// TIA Portal V17 export
// export: Created 2025-03-05T08:02:58.0476046Z, ExportSetting WithDefaults, DisplayName Totally Integrated Automation Portal, DisplayVersion V17 Update 8, DisplayName TIA Portal Openness, DisplayVersion V17 Update 8, DisplayName TIA Portal Version Control Interface, DisplayVersion V17, DisplayName SINAMICS Startdrive Advanced, DisplayVersion V17 SP2, DisplayName SINAMICS Startdrive G110M, G120, G120C, G120D, G120P, G115D, DisplayVersion V17 SP2, DisplayName SINAMICS Startdrive G130, G150, S120, S150, SINAMICS MV, S210, DisplayVersion V17 SP2, DisplayName STEP 7 Professional, DisplayVersion V17 Update 8, DisplayName SINUMERIK ONE STEP 7 Toolbox, DisplayVersion V17 Update 12, DisplayName SINUMERIK 840D sl STEP 7 Toolbox, DisplayVersion V17 Update 12, DisplayName STEP 7 Safety, DisplayVersion V17 Update 6, DisplayName WinCC Advanced, DisplayVersion V17 Update 8
FUNCTION "FC16702_OPC_UA_MASTER_POWDER_DATA_UPDATE" : Void   // FC16702, LAD
{ S7_Optimized_Access := 'TRUE' }
VERSION : 0.1
// stored: AutoNumber false, IsIECCheckEnabled false, SetENOAutomatically false, UDAEnableTagReadback false
   VAR_TEMP
      CURRENT_1 : Real;
      CURRENT_2 : Real;
      CURRENT_3 : Real;
      CURRENT_4 : Real;
      CURRENT_5 : Real;
      CURRENT_6 : Real;
      CURRENT_7 : Real;
      CURRENT_8 : Real;
      CURRENT_9 : Real;
      CURRENT_10 : Real;
   END_VAR
BEGIN

REGION Network 1: <<<<<<<<<<<<<<<<<<<< OPC UA MASTER POWDER >>>>>>>>>>>>>>>>>>>>
END_REGION

REGION Network 2: <<<<<<<<<<<<<< GENERAL >>>>>>>>>>>>>>>>>>>>
END_REGION

REGION Network 3: GENERAL INFO
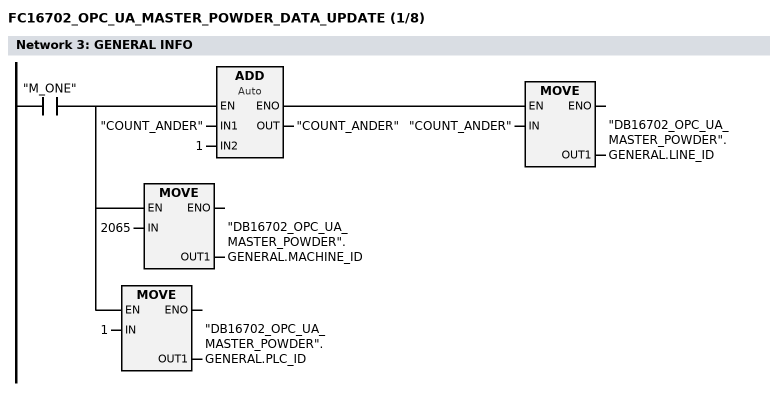
   RUNG wire#powerrail
      Contact( "M_ONE" )
      wire#w1
      Add(in1 := "COUNT_ANDER", in2 := 1, out => "COUNT_ANDER")
      Move(in := "COUNT_ANDER", out1 => "DB16702_OPC_UA_MASTER_POWDER".GENERAL.LINE_ID)
   END_RUNG
   RUNG wire#w1
      Move(in := 2065, out1 => "DB16702_OPC_UA_MASTER_POWDER".GENERAL.MACHINE_ID)
   END_RUNG
   RUNG wire#w1
      Move(in := 1, out1 => "DB16702_OPC_UA_MASTER_POWDER".GENERAL.PLC_ID)
   END_RUNG
   // the same network as SCL:
   IF "M_ONE" THEN
       "COUNT_ANDER" := "COUNT_ANDER" + 1;
       "DB16702_OPC_UA_MASTER_POWDER".GENERAL.LINE_ID := "COUNT_ANDER";
       "DB16702_OPC_UA_MASTER_POWDER".GENERAL.MACHINE_ID := 2065;
       "DB16702_OPC_UA_MASTER_POWDER".GENERAL.PLC_ID := 1;
   END_IF;
END_REGION

REGION Network 4: <<<<<<<<<<<<<< UNIT 01 >>>>>>>>>>>>>>>>>>>>
END_REGION

REGION Network 5: HOPPER 1 UNIT 01
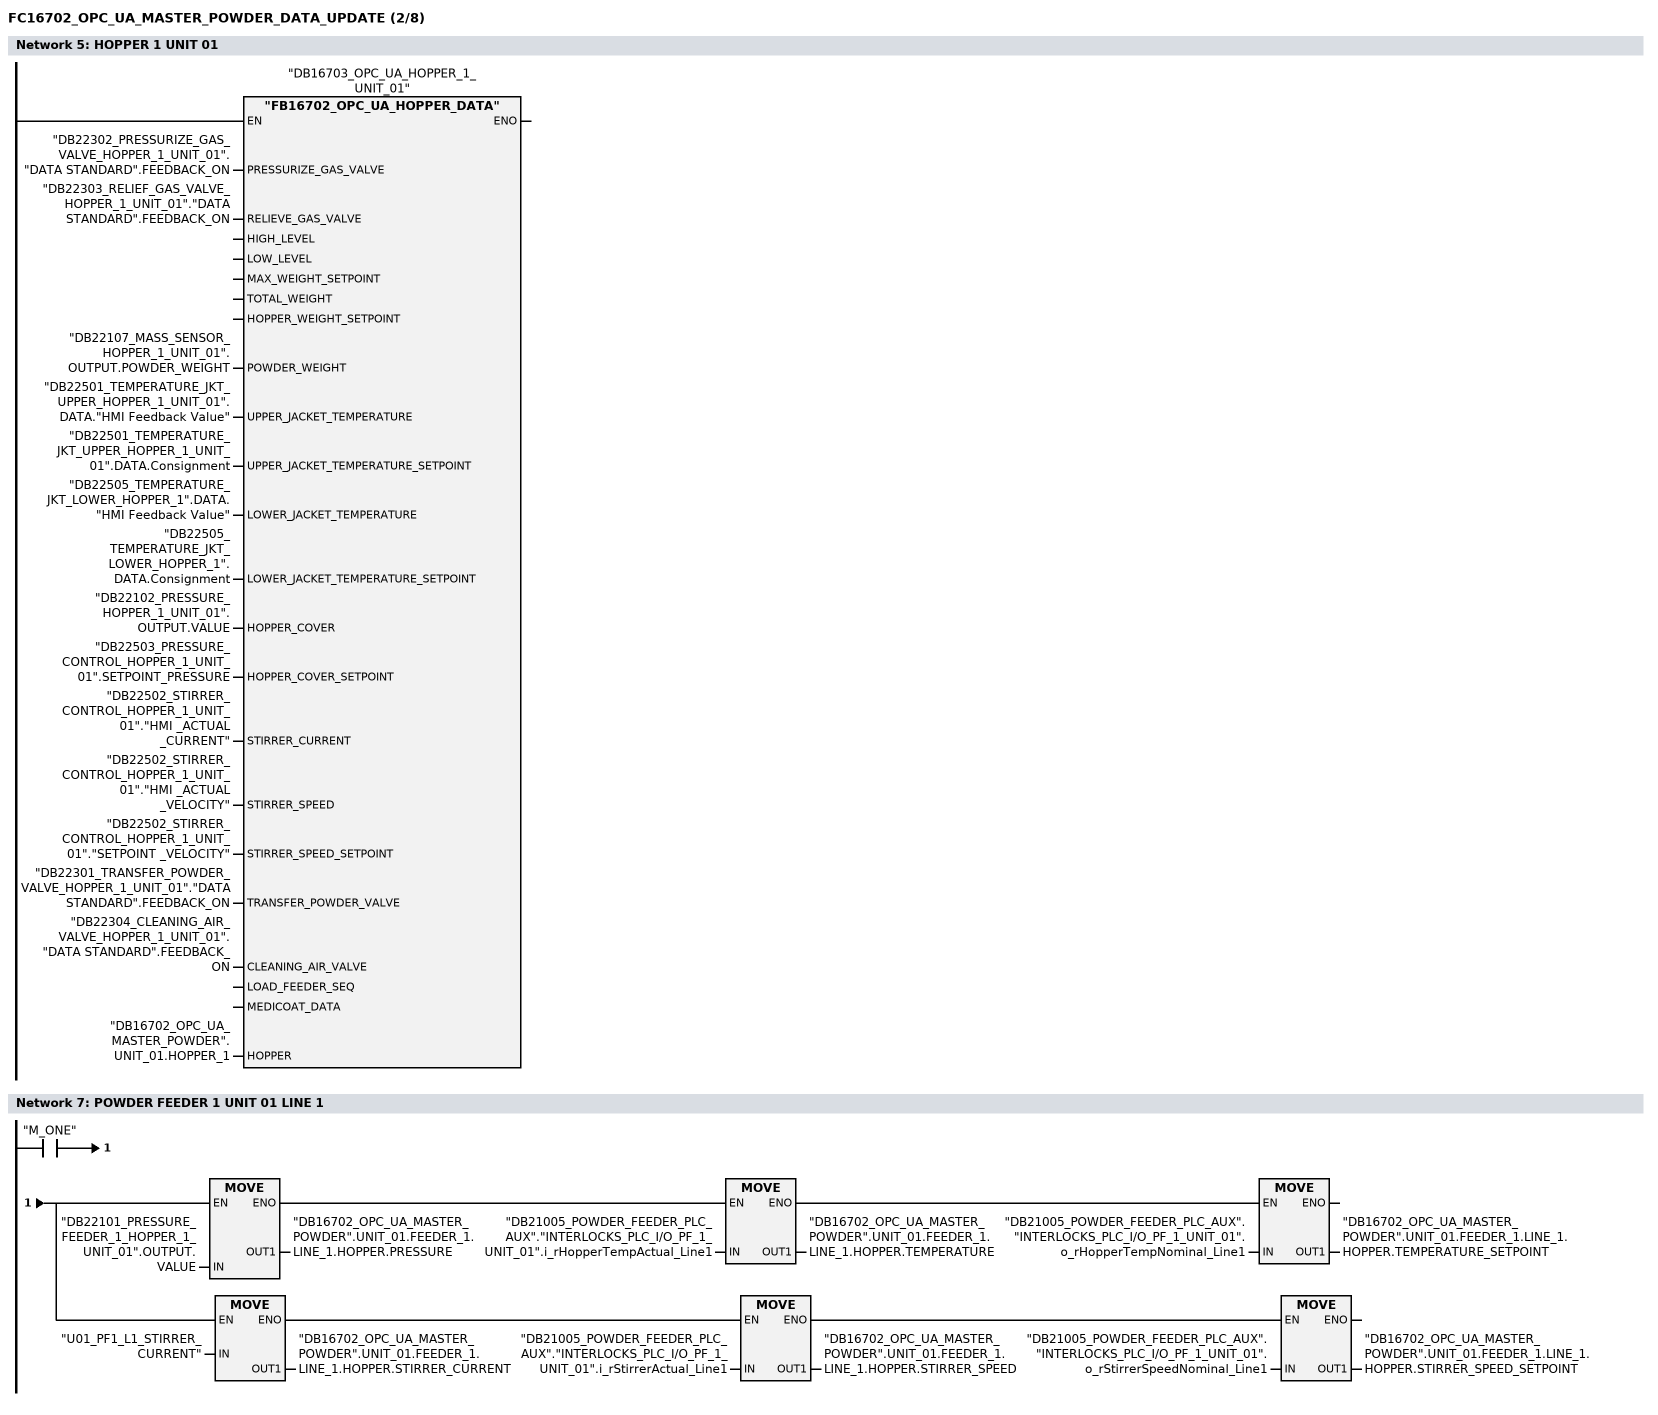
   RUNG wire#powerrail
      "DB16703_OPC_UA_HOPPER_1_UNIT_01"(PRESSURIZE_GAS_VALVE := "DB22302_PRESSURIZE_GAS_VALVE_HOPPER_1_UNIT_01"."DATA STANDARD".FEEDBACK_ON, RELIEVE_GAS_VALVE := "DB22303_RELIEF_GAS_VALVE_HOPPER_1_UNIT_01"."DATA STANDARD".FEEDBACK_ON, HIGH_LEVEL :=, LOW_LEVEL :=, MAX_WEIGHT_SETPOINT :=, TOTAL_WEIGHT :=, HOPPER_WEIGHT_SETPOINT :=, POWDER_WEIGHT := "DB22107_MASS_SENSOR_HOPPER_1_UNIT_01".OUTPUT.POWDER_WEIGHT, UPPER_JACKET_TEMPERATURE := "DB22501_TEMPERATURE_JKT_UPPER_HOPPER_1_UNIT_01".DATA."HMI Feedback Value", UPPER_JACKET_TEMPERATURE_SETPOINT := "DB22501_TEMPERATURE_JKT_UPPER_HOPPER_1_UNIT_01".DATA.Consignment, LOWER_JACKET_TEMPERATURE := "DB22505_TEMPERATURE_JKT_LOWER_HOPPER_1".DATA."HMI Feedback Value", LOWER_JACKET_TEMPERATURE_SETPOINT := "DB22505_TEMPERATURE_JKT_LOWER_HOPPER_1".DATA.Consignment, HOPPER_COVER := "DB22102_PRESSURE_HOPPER_1_UNIT_01".OUTPUT.VALUE, HOPPER_COVER_SETPOINT := "DB22503_PRESSURE_CONTROL_HOPPER_1_UNIT_01".SETPOINT_PRESSURE, STIRRER_CURRENT := "DB22502_STIRRER_CONTROL_HOPPER_1_UNIT_01"."HMI _ACTUAL _CURRENT", STIRRER_SPEED := "DB22502_STIRRER_CONTROL_HOPPER_1_UNIT_01"."HMI _ACTUAL _VELOCITY", STIRRER_SPEED_SETPOINT := "DB22502_STIRRER_CONTROL_HOPPER_1_UNIT_01"."SETPOINT _VELOCITY", TRANSFER_POWDER_VALVE := "DB22301_TRANSFER_POWDER_VALVE_HOPPER_1_UNIT_01"."DATA STANDARD".FEEDBACK_ON, CLEANING_AIR_VALVE := "DB22304_CLEANING_AIR_VALVE_HOPPER_1_UNIT_01"."DATA STANDARD".FEEDBACK_ON, LOAD_FEEDER_SEQ :=, MEDICOAT_DATA :=, HOPPER := "DB16702_OPC_UA_MASTER_POWDER".UNIT_01.HOPPER_1)
   END_RUNG
   // the same network as SCL:
   "DB16703_OPC_UA_HOPPER_1_UNIT_01"(PRESSURIZE_GAS_VALVE := "DB22302_PRESSURIZE_GAS_VALVE_HOPPER_1_UNIT_01"."DATA STANDARD".FEEDBACK_ON,   // "FB16702_OPC_UA_HOPPER_DATA"
                           RELIEVE_GAS_VALVE := "DB22303_RELIEF_GAS_VALVE_HOPPER_1_UNIT_01"."DATA STANDARD".FEEDBACK_ON,
                           POWDER_WEIGHT := "DB22107_MASS_SENSOR_HOPPER_1_UNIT_01".OUTPUT.POWDER_WEIGHT,
                           UPPER_JACKET_TEMPERATURE := "DB22501_TEMPERATURE_JKT_UPPER_HOPPER_1_UNIT_01".DATA."HMI Feedback Value",
                           UPPER_JACKET_TEMPERATURE_SETPOINT := "DB22501_TEMPERATURE_JKT_UPPER_HOPPER_1_UNIT_01".DATA.Consignment,
                           LOWER_JACKET_TEMPERATURE := "DB22505_TEMPERATURE_JKT_LOWER_HOPPER_1".DATA."HMI Feedback Value",
                           LOWER_JACKET_TEMPERATURE_SETPOINT := "DB22505_TEMPERATURE_JKT_LOWER_HOPPER_1".DATA.Consignment,
                           HOPPER_COVER := "DB22102_PRESSURE_HOPPER_1_UNIT_01".OUTPUT.VALUE,
                           HOPPER_COVER_SETPOINT := "DB22503_PRESSURE_CONTROL_HOPPER_1_UNIT_01".SETPOINT_PRESSURE,
                           STIRRER_CURRENT := "DB22502_STIRRER_CONTROL_HOPPER_1_UNIT_01"."HMI _ACTUAL _CURRENT",
                           STIRRER_SPEED := "DB22502_STIRRER_CONTROL_HOPPER_1_UNIT_01"."HMI _ACTUAL _VELOCITY",
                           STIRRER_SPEED_SETPOINT := "DB22502_STIRRER_CONTROL_HOPPER_1_UNIT_01"."SETPOINT _VELOCITY",
                           TRANSFER_POWDER_VALVE := "DB22301_TRANSFER_POWDER_VALVE_HOPPER_1_UNIT_01"."DATA STANDARD".FEEDBACK_ON,
                           CLEANING_AIR_VALVE := "DB22304_CLEANING_AIR_VALVE_HOPPER_1_UNIT_01"."DATA STANDARD".FEEDBACK_ON,
                           HOPPER := "DB16702_OPC_UA_MASTER_POWDER".UNIT_01.HOPPER_1);
END_REGION

REGION Network 6: HOPPER 2 UNIT 01
END_REGION

REGION Network 7: POWDER FEEDER 1 UNIT 01 LINE 1
   RUNG wire#powerrail
      Contact( "M_ONE" )
      wire#w1
      Move(in := "DB22101_PRESSURE_FEEDER_1_HOPPER_1_UNIT_01".OUTPUT.VALUE, out1 => "DB16702_OPC_UA_MASTER_POWDER".UNIT_01.FEEDER_1.LINE_1.HOPPER.PRESSURE)
      Move(in := "DB21005_POWDER_FEEDER_PLC_AUX"."INTERLOCKS_PLC_I/O_PF_1_UNIT_01".i_rHopperTempActual_Line1, out1 => "DB16702_OPC_UA_MASTER_POWDER".UNIT_01.FEEDER_1.LINE_1.HOPPER.TEMPERATURE)
      Move(in := "DB21005_POWDER_FEEDER_PLC_AUX"."INTERLOCKS_PLC_I/O_PF_1_UNIT_01".o_rHopperTempNominal_Line1, out1 => "DB16702_OPC_UA_MASTER_POWDER".UNIT_01.FEEDER_1.LINE_1.HOPPER.TEMPERATURE_SETPOINT)
   END_RUNG
   RUNG wire#w1
      Move(in := "U01_PF1_L1_STIRRER_CURRENT", out1 => "DB16702_OPC_UA_MASTER_POWDER".UNIT_01.FEEDER_1.LINE_1.HOPPER.STIRRER_CURRENT)
      Move(in := "DB21005_POWDER_FEEDER_PLC_AUX"."INTERLOCKS_PLC_I/O_PF_1_UNIT_01".i_rStirrerActual_Line1, out1 => "DB16702_OPC_UA_MASTER_POWDER".UNIT_01.FEEDER_1.LINE_1.HOPPER.STIRRER_SPEED)
      Move(in := "DB21005_POWDER_FEEDER_PLC_AUX"."INTERLOCKS_PLC_I/O_PF_1_UNIT_01".o_rStirrerSpeedNominal_Line1, out1 => "DB16702_OPC_UA_MASTER_POWDER".UNIT_01.FEEDER_1.LINE_1.HOPPER.STIRRER_SPEED_SETPOINT)
   END_RUNG
   // the same network as SCL:
   IF "M_ONE" THEN
       "DB16702_OPC_UA_MASTER_POWDER".UNIT_01.FEEDER_1.LINE_1.HOPPER.PRESSURE := "DB22101_PRESSURE_FEEDER_1_HOPPER_1_UNIT_01".OUTPUT.VALUE;
       "DB16702_OPC_UA_MASTER_POWDER".UNIT_01.FEEDER_1.LINE_1.HOPPER.TEMPERATURE := "DB21005_POWDER_FEEDER_PLC_AUX"."INTERLOCKS_PLC_I/O_PF_1_UNIT_01".i_rHopperTempActual_Line1;
       "DB16702_OPC_UA_MASTER_POWDER".UNIT_01.FEEDER_1.LINE_1.HOPPER.TEMPERATURE_SETPOINT := "DB21005_POWDER_FEEDER_PLC_AUX"."INTERLOCKS_PLC_I/O_PF_1_UNIT_01".o_rHopperTempNominal_Line1;
       "DB16702_OPC_UA_MASTER_POWDER".UNIT_01.FEEDER_1.LINE_1.HOPPER.STIRRER_CURRENT := "U01_PF1_L1_STIRRER_CURRENT";
       "DB16702_OPC_UA_MASTER_POWDER".UNIT_01.FEEDER_1.LINE_1.HOPPER.STIRRER_SPEED := "DB21005_POWDER_FEEDER_PLC_AUX"."INTERLOCKS_PLC_I/O_PF_1_UNIT_01".i_rStirrerActual_Line1;
       "DB16702_OPC_UA_MASTER_POWDER".UNIT_01.FEEDER_1.LINE_1.HOPPER.STIRRER_SPEED_SETPOINT := "DB21005_POWDER_FEEDER_PLC_AUX"."INTERLOCKS_PLC_I/O_PF_1_UNIT_01".o_rStirrerSpeedNominal_Line1;
   END_IF;
END_REGION

REGION Network 8: POWDER FEEDER 1 UNIT 01 LINE 1 DISK
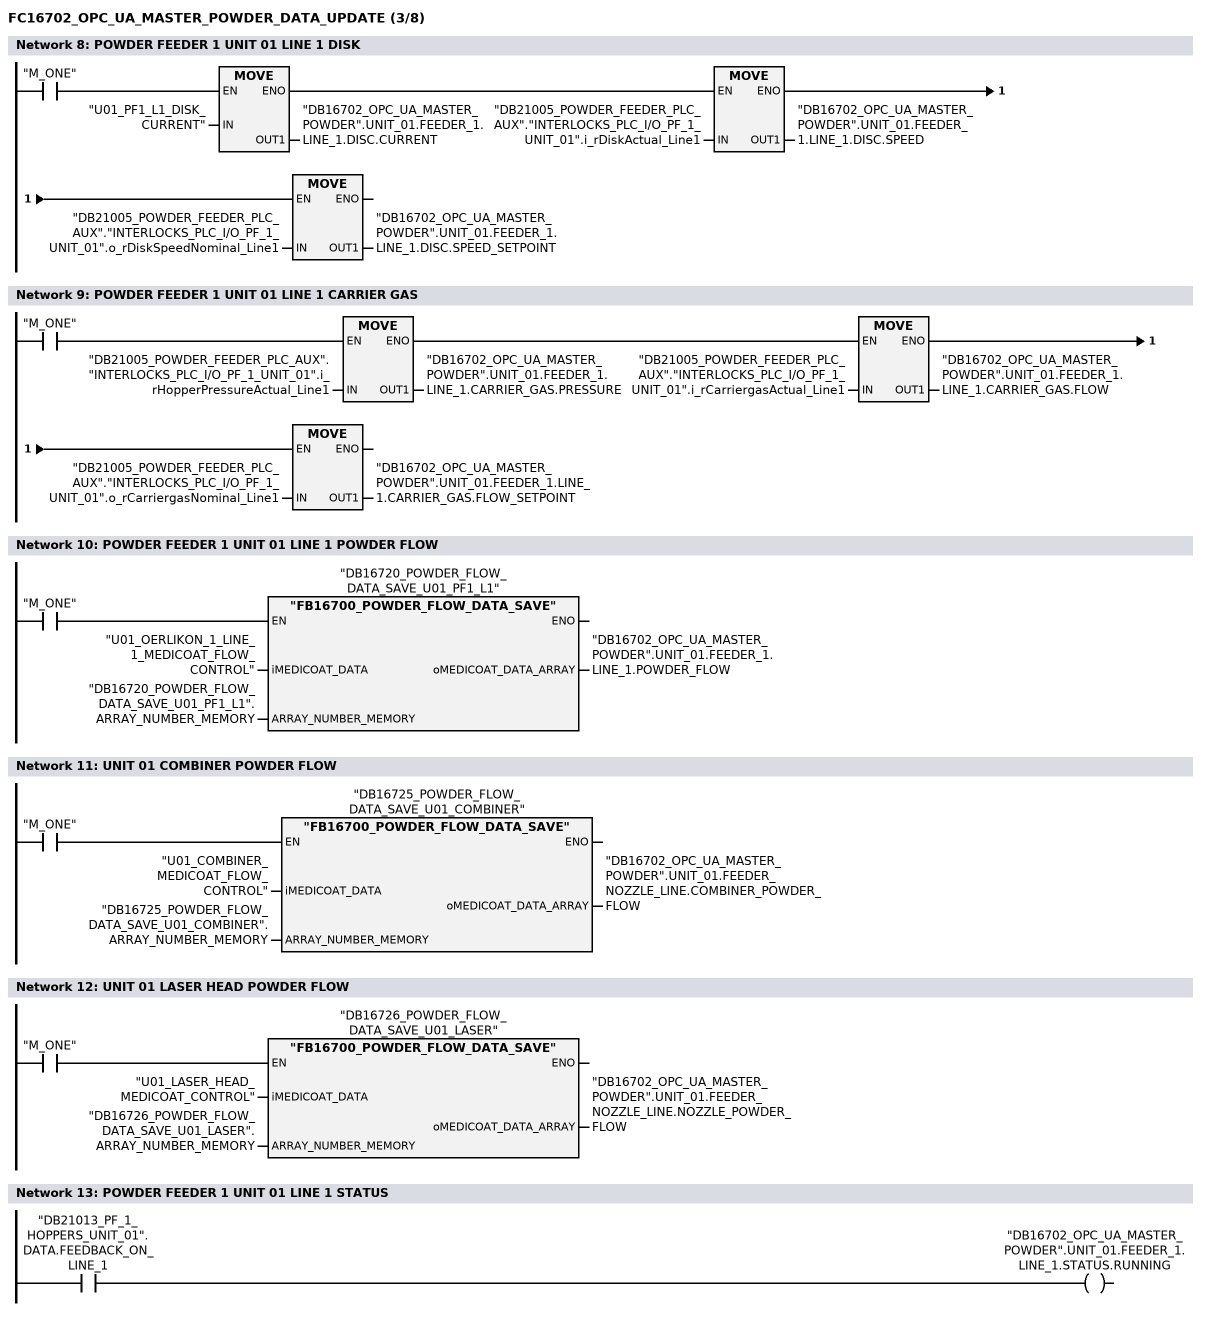
   RUNG wire#powerrail
      Contact( "M_ONE" )
      Move(in := "U01_PF1_L1_DISK_CURRENT", out1 => "DB16702_OPC_UA_MASTER_POWDER".UNIT_01.FEEDER_1.LINE_1.DISC.CURRENT)
      Move(in := "DB21005_POWDER_FEEDER_PLC_AUX"."INTERLOCKS_PLC_I/O_PF_1_UNIT_01".i_rDiskActual_Line1, out1 => "DB16702_OPC_UA_MASTER_POWDER".UNIT_01.FEEDER_1.LINE_1.DISC.SPEED)
      Move(in := "DB21005_POWDER_FEEDER_PLC_AUX"."INTERLOCKS_PLC_I/O_PF_1_UNIT_01".o_rDiskSpeedNominal_Line1, out1 => "DB16702_OPC_UA_MASTER_POWDER".UNIT_01.FEEDER_1.LINE_1.DISC.SPEED_SETPOINT)
   END_RUNG
   // the same network as SCL:
   IF "M_ONE" THEN
       "DB16702_OPC_UA_MASTER_POWDER".UNIT_01.FEEDER_1.LINE_1.DISC.CURRENT := "U01_PF1_L1_DISK_CURRENT";
       "DB16702_OPC_UA_MASTER_POWDER".UNIT_01.FEEDER_1.LINE_1.DISC.SPEED := "DB21005_POWDER_FEEDER_PLC_AUX"."INTERLOCKS_PLC_I/O_PF_1_UNIT_01".i_rDiskActual_Line1;
       "DB16702_OPC_UA_MASTER_POWDER".UNIT_01.FEEDER_1.LINE_1.DISC.SPEED_SETPOINT := "DB21005_POWDER_FEEDER_PLC_AUX"."INTERLOCKS_PLC_I/O_PF_1_UNIT_01".o_rDiskSpeedNominal_Line1;
   END_IF;
END_REGION

REGION Network 9: POWDER FEEDER 1 UNIT 01 LINE 1 CARRIER GAS
   RUNG wire#powerrail
      Contact( "M_ONE" )
      Move(in := "DB21005_POWDER_FEEDER_PLC_AUX"."INTERLOCKS_PLC_I/O_PF_1_UNIT_01".i_rHopperPressureActual_Line1, out1 => "DB16702_OPC_UA_MASTER_POWDER".UNIT_01.FEEDER_1.LINE_1.CARRIER_GAS.PRESSURE)
      Move(in := "DB21005_POWDER_FEEDER_PLC_AUX"."INTERLOCKS_PLC_I/O_PF_1_UNIT_01".i_rCarriergasActual_Line1, out1 => "DB16702_OPC_UA_MASTER_POWDER".UNIT_01.FEEDER_1.LINE_1.CARRIER_GAS.FLOW)
      Move(in := "DB21005_POWDER_FEEDER_PLC_AUX"."INTERLOCKS_PLC_I/O_PF_1_UNIT_01".o_rCarriergasNominal_Line1, out1 => "DB16702_OPC_UA_MASTER_POWDER".UNIT_01.FEEDER_1.LINE_1.CARRIER_GAS.FLOW_SETPOINT)
   END_RUNG
   // the same network as SCL:
   IF "M_ONE" THEN
       "DB16702_OPC_UA_MASTER_POWDER".UNIT_01.FEEDER_1.LINE_1.CARRIER_GAS.PRESSURE := "DB21005_POWDER_FEEDER_PLC_AUX"."INTERLOCKS_PLC_I/O_PF_1_UNIT_01".i_rHopperPressureActual_Line1;
       "DB16702_OPC_UA_MASTER_POWDER".UNIT_01.FEEDER_1.LINE_1.CARRIER_GAS.FLOW := "DB21005_POWDER_FEEDER_PLC_AUX"."INTERLOCKS_PLC_I/O_PF_1_UNIT_01".i_rCarriergasActual_Line1;
       "DB16702_OPC_UA_MASTER_POWDER".UNIT_01.FEEDER_1.LINE_1.CARRIER_GAS.FLOW_SETPOINT := "DB21005_POWDER_FEEDER_PLC_AUX"."INTERLOCKS_PLC_I/O_PF_1_UNIT_01".o_rCarriergasNominal_Line1;
   END_IF;
END_REGION

REGION Network 10: POWDER FEEDER 1 UNIT 01 LINE 1 POWDER FLOW
   RUNG wire#powerrail
      Contact( "M_ONE" )
      "DB16720_POWDER_FLOW_DATA_SAVE_U01_PF1_L1"(iMEDICOAT_DATA := "U01_OERLIKON_1_LINE_1_MEDICOAT_FLOW_CONTROL", ARRAY_NUMBER_MEMORY := "DB16720_POWDER_FLOW_DATA_SAVE_U01_PF1_L1".ARRAY_NUMBER_MEMORY, oMEDICOAT_DATA_ARRAY => "DB16702_OPC_UA_MASTER_POWDER".UNIT_01.FEEDER_1.LINE_1.POWDER_FLOW)
   END_RUNG
   // the same network as SCL:
   IF "M_ONE" THEN
       "DB16720_POWDER_FLOW_DATA_SAVE_U01_PF1_L1"(iMEDICOAT_DATA := "U01_OERLIKON_1_LINE_1_MEDICOAT_FLOW_CONTROL",   // "FB16700_POWDER_FLOW_DATA_SAVE"
                               ARRAY_NUMBER_MEMORY := "DB16720_POWDER_FLOW_DATA_SAVE_U01_PF1_L1".ARRAY_NUMBER_MEMORY,
                               oMEDICOAT_DATA_ARRAY => "DB16702_OPC_UA_MASTER_POWDER".UNIT_01.FEEDER_1.LINE_1.POWDER_FLOW);
   END_IF;
END_REGION

REGION Network 11: UNIT 01 COMBINER POWDER FLOW
   RUNG wire#powerrail
      Contact( "M_ONE" )
      "DB16725_POWDER_FLOW_DATA_SAVE_U01_COMBINER"(iMEDICOAT_DATA := "U01_COMBINER_MEDICOAT_FLOW_CONTROL", ARRAY_NUMBER_MEMORY := "DB16725_POWDER_FLOW_DATA_SAVE_U01_COMBINER".ARRAY_NUMBER_MEMORY, oMEDICOAT_DATA_ARRAY => "DB16702_OPC_UA_MASTER_POWDER".UNIT_01.FEEDER_NOZZLE_LINE.COMBINER_POWDER_FLOW)
   END_RUNG
   // the same network as SCL:
   IF "M_ONE" THEN
       "DB16725_POWDER_FLOW_DATA_SAVE_U01_COMBINER"(iMEDICOAT_DATA := "U01_COMBINER_MEDICOAT_FLOW_CONTROL",   // "FB16700_POWDER_FLOW_DATA_SAVE"
                               ARRAY_NUMBER_MEMORY := "DB16725_POWDER_FLOW_DATA_SAVE_U01_COMBINER".ARRAY_NUMBER_MEMORY,
                               oMEDICOAT_DATA_ARRAY => "DB16702_OPC_UA_MASTER_POWDER".UNIT_01.FEEDER_NOZZLE_LINE.COMBINER_POWDER_FLOW);
   END_IF;
END_REGION

REGION Network 12: UNIT 01 LASER HEAD POWDER FLOW
   RUNG wire#powerrail
      Contact( "M_ONE" )
      "DB16726_POWDER_FLOW_DATA_SAVE_U01_LASER"(iMEDICOAT_DATA := "U01_LASER_HEAD_MEDICOAT_CONTROL", ARRAY_NUMBER_MEMORY := "DB16726_POWDER_FLOW_DATA_SAVE_U01_LASER".ARRAY_NUMBER_MEMORY, oMEDICOAT_DATA_ARRAY => "DB16702_OPC_UA_MASTER_POWDER".UNIT_01.FEEDER_NOZZLE_LINE.NOZZLE_POWDER_FLOW)
   END_RUNG
   // the same network as SCL:
   IF "M_ONE" THEN
       "DB16726_POWDER_FLOW_DATA_SAVE_U01_LASER"(iMEDICOAT_DATA := "U01_LASER_HEAD_MEDICOAT_CONTROL",   // "FB16700_POWDER_FLOW_DATA_SAVE"
                               ARRAY_NUMBER_MEMORY := "DB16726_POWDER_FLOW_DATA_SAVE_U01_LASER".ARRAY_NUMBER_MEMORY,
                               oMEDICOAT_DATA_ARRAY => "DB16702_OPC_UA_MASTER_POWDER".UNIT_01.FEEDER_NOZZLE_LINE.NOZZLE_POWDER_FLOW);
   END_IF;
END_REGION

REGION Network 13: POWDER FEEDER 1 UNIT 01 LINE 1 STATUS
   RUNG wire#powerrail
      Contact( "DB21013_PF_1_HOPPERS_UNIT_01".DATA.FEEDBACK_ON_LINE_1 )
      Coil( "DB16702_OPC_UA_MASTER_POWDER".UNIT_01.FEEDER_1.LINE_1.STATUS.RUNNING )
   END_RUNG
   // the same network as SCL:
   "DB16702_OPC_UA_MASTER_POWDER".UNIT_01.FEEDER_1.LINE_1.STATUS.RUNNING := "DB21013_PF_1_HOPPERS_UNIT_01".DATA.FEEDBACK_ON_LINE_1;
END_REGION

REGION Network 14: POWDER FEEDER 1 UNIT 01 LINE 2 HOPPER
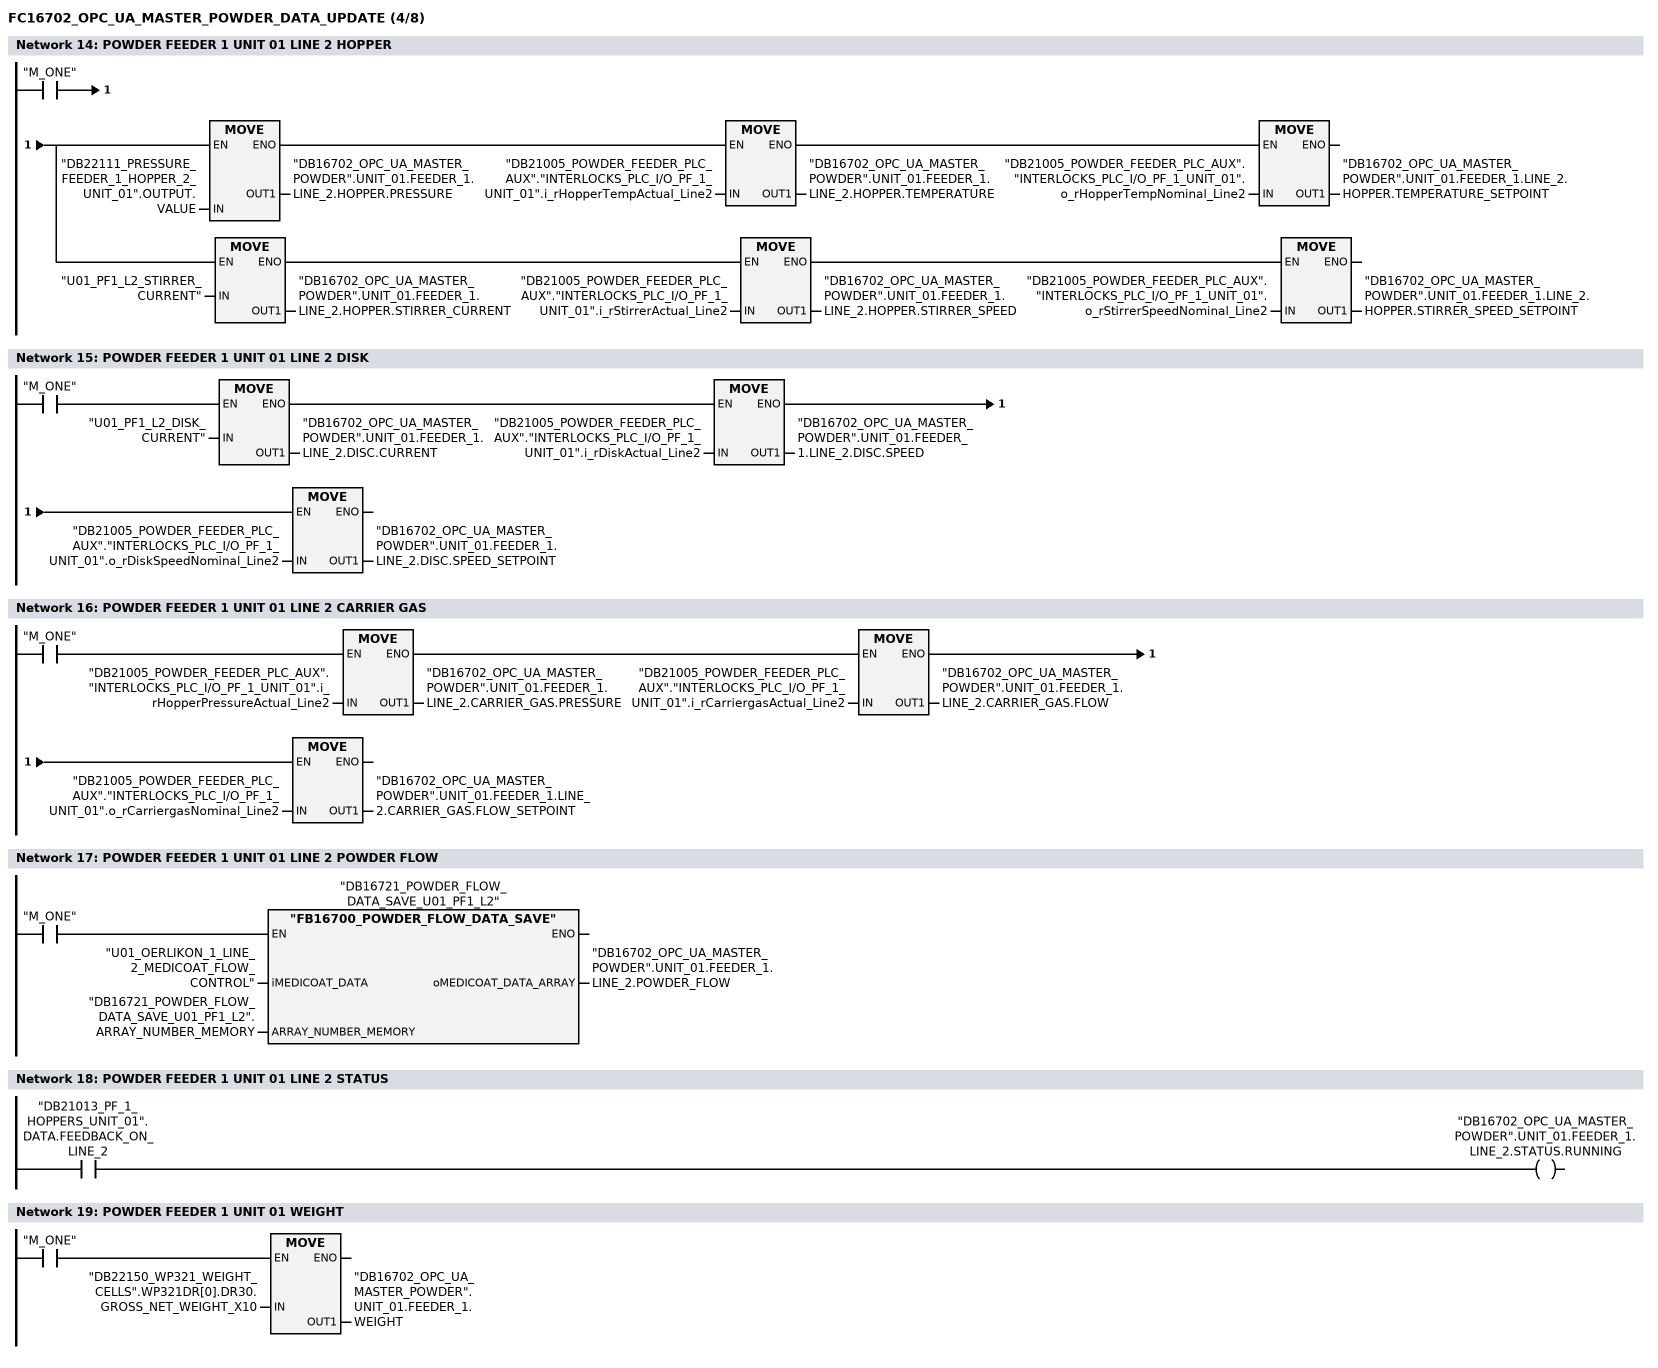
   RUNG wire#powerrail
      Contact( "M_ONE" )
      wire#w1
      Move(in := "DB22111_PRESSURE_FEEDER_1_HOPPER_2_UNIT_01".OUTPUT.VALUE, out1 => "DB16702_OPC_UA_MASTER_POWDER".UNIT_01.FEEDER_1.LINE_2.HOPPER.PRESSURE)
      Move(in := "DB21005_POWDER_FEEDER_PLC_AUX"."INTERLOCKS_PLC_I/O_PF_1_UNIT_01".i_rHopperTempActual_Line2, out1 => "DB16702_OPC_UA_MASTER_POWDER".UNIT_01.FEEDER_1.LINE_2.HOPPER.TEMPERATURE)
      Move(in := "DB21005_POWDER_FEEDER_PLC_AUX"."INTERLOCKS_PLC_I/O_PF_1_UNIT_01".o_rHopperTempNominal_Line2, out1 => "DB16702_OPC_UA_MASTER_POWDER".UNIT_01.FEEDER_1.LINE_2.HOPPER.TEMPERATURE_SETPOINT)
   END_RUNG
   RUNG wire#w1
      Move(in := "U01_PF1_L2_STIRRER_CURRENT", out1 => "DB16702_OPC_UA_MASTER_POWDER".UNIT_01.FEEDER_1.LINE_2.HOPPER.STIRRER_CURRENT)
      Move(in := "DB21005_POWDER_FEEDER_PLC_AUX"."INTERLOCKS_PLC_I/O_PF_1_UNIT_01".i_rStirrerActual_Line2, out1 => "DB16702_OPC_UA_MASTER_POWDER".UNIT_01.FEEDER_1.LINE_2.HOPPER.STIRRER_SPEED)
      Move(in := "DB21005_POWDER_FEEDER_PLC_AUX"."INTERLOCKS_PLC_I/O_PF_1_UNIT_01".o_rStirrerSpeedNominal_Line2, out1 => "DB16702_OPC_UA_MASTER_POWDER".UNIT_01.FEEDER_1.LINE_2.HOPPER.STIRRER_SPEED_SETPOINT)
   END_RUNG
   // the same network as SCL:
   IF "M_ONE" THEN
       "DB16702_OPC_UA_MASTER_POWDER".UNIT_01.FEEDER_1.LINE_2.HOPPER.PRESSURE := "DB22111_PRESSURE_FEEDER_1_HOPPER_2_UNIT_01".OUTPUT.VALUE;
       "DB16702_OPC_UA_MASTER_POWDER".UNIT_01.FEEDER_1.LINE_2.HOPPER.TEMPERATURE := "DB21005_POWDER_FEEDER_PLC_AUX"."INTERLOCKS_PLC_I/O_PF_1_UNIT_01".i_rHopperTempActual_Line2;
       "DB16702_OPC_UA_MASTER_POWDER".UNIT_01.FEEDER_1.LINE_2.HOPPER.TEMPERATURE_SETPOINT := "DB21005_POWDER_FEEDER_PLC_AUX"."INTERLOCKS_PLC_I/O_PF_1_UNIT_01".o_rHopperTempNominal_Line2;
       "DB16702_OPC_UA_MASTER_POWDER".UNIT_01.FEEDER_1.LINE_2.HOPPER.STIRRER_CURRENT := "U01_PF1_L2_STIRRER_CURRENT";
       "DB16702_OPC_UA_MASTER_POWDER".UNIT_01.FEEDER_1.LINE_2.HOPPER.STIRRER_SPEED := "DB21005_POWDER_FEEDER_PLC_AUX"."INTERLOCKS_PLC_I/O_PF_1_UNIT_01".i_rStirrerActual_Line2;
       "DB16702_OPC_UA_MASTER_POWDER".UNIT_01.FEEDER_1.LINE_2.HOPPER.STIRRER_SPEED_SETPOINT := "DB21005_POWDER_FEEDER_PLC_AUX"."INTERLOCKS_PLC_I/O_PF_1_UNIT_01".o_rStirrerSpeedNominal_Line2;
   END_IF;
END_REGION

REGION Network 15: POWDER FEEDER 1 UNIT 01 LINE 2 DISK
   RUNG wire#powerrail
      Contact( "M_ONE" )
      Move(in := "U01_PF1_L2_DISK_CURRENT", out1 => "DB16702_OPC_UA_MASTER_POWDER".UNIT_01.FEEDER_1.LINE_2.DISC.CURRENT)
      Move(in := "DB21005_POWDER_FEEDER_PLC_AUX"."INTERLOCKS_PLC_I/O_PF_1_UNIT_01".i_rDiskActual_Line2, out1 => "DB16702_OPC_UA_MASTER_POWDER".UNIT_01.FEEDER_1.LINE_2.DISC.SPEED)
      Move(in := "DB21005_POWDER_FEEDER_PLC_AUX"."INTERLOCKS_PLC_I/O_PF_1_UNIT_01".o_rDiskSpeedNominal_Line2, out1 => "DB16702_OPC_UA_MASTER_POWDER".UNIT_01.FEEDER_1.LINE_2.DISC.SPEED_SETPOINT)
   END_RUNG
   // the same network as SCL:
   IF "M_ONE" THEN
       "DB16702_OPC_UA_MASTER_POWDER".UNIT_01.FEEDER_1.LINE_2.DISC.CURRENT := "U01_PF1_L2_DISK_CURRENT";
       "DB16702_OPC_UA_MASTER_POWDER".UNIT_01.FEEDER_1.LINE_2.DISC.SPEED := "DB21005_POWDER_FEEDER_PLC_AUX"."INTERLOCKS_PLC_I/O_PF_1_UNIT_01".i_rDiskActual_Line2;
       "DB16702_OPC_UA_MASTER_POWDER".UNIT_01.FEEDER_1.LINE_2.DISC.SPEED_SETPOINT := "DB21005_POWDER_FEEDER_PLC_AUX"."INTERLOCKS_PLC_I/O_PF_1_UNIT_01".o_rDiskSpeedNominal_Line2;
   END_IF;
END_REGION

REGION Network 16: POWDER FEEDER 1 UNIT 01 LINE 2 CARRIER GAS
   RUNG wire#powerrail
      Contact( "M_ONE" )
      Move(in := "DB21005_POWDER_FEEDER_PLC_AUX"."INTERLOCKS_PLC_I/O_PF_1_UNIT_01".i_rHopperPressureActual_Line2, out1 => "DB16702_OPC_UA_MASTER_POWDER".UNIT_01.FEEDER_1.LINE_2.CARRIER_GAS.PRESSURE)
      Move(in := "DB21005_POWDER_FEEDER_PLC_AUX"."INTERLOCKS_PLC_I/O_PF_1_UNIT_01".i_rCarriergasActual_Line2, out1 => "DB16702_OPC_UA_MASTER_POWDER".UNIT_01.FEEDER_1.LINE_2.CARRIER_GAS.FLOW)
      Move(in := "DB21005_POWDER_FEEDER_PLC_AUX"."INTERLOCKS_PLC_I/O_PF_1_UNIT_01".o_rCarriergasNominal_Line2, out1 => "DB16702_OPC_UA_MASTER_POWDER".UNIT_01.FEEDER_1.LINE_2.CARRIER_GAS.FLOW_SETPOINT)
   END_RUNG
   // the same network as SCL:
   IF "M_ONE" THEN
       "DB16702_OPC_UA_MASTER_POWDER".UNIT_01.FEEDER_1.LINE_2.CARRIER_GAS.PRESSURE := "DB21005_POWDER_FEEDER_PLC_AUX"."INTERLOCKS_PLC_I/O_PF_1_UNIT_01".i_rHopperPressureActual_Line2;
       "DB16702_OPC_UA_MASTER_POWDER".UNIT_01.FEEDER_1.LINE_2.CARRIER_GAS.FLOW := "DB21005_POWDER_FEEDER_PLC_AUX"."INTERLOCKS_PLC_I/O_PF_1_UNIT_01".i_rCarriergasActual_Line2;
       "DB16702_OPC_UA_MASTER_POWDER".UNIT_01.FEEDER_1.LINE_2.CARRIER_GAS.FLOW_SETPOINT := "DB21005_POWDER_FEEDER_PLC_AUX"."INTERLOCKS_PLC_I/O_PF_1_UNIT_01".o_rCarriergasNominal_Line2;
   END_IF;
END_REGION

REGION Network 17: POWDER FEEDER 1 UNIT 01 LINE 2 POWDER FLOW
   RUNG wire#powerrail
      Contact( "M_ONE" )
      "DB16721_POWDER_FLOW_DATA_SAVE_U01_PF1_L2"(iMEDICOAT_DATA := "U01_OERLIKON_1_LINE_2_MEDICOAT_FLOW_CONTROL", ARRAY_NUMBER_MEMORY := "DB16721_POWDER_FLOW_DATA_SAVE_U01_PF1_L2".ARRAY_NUMBER_MEMORY, oMEDICOAT_DATA_ARRAY => "DB16702_OPC_UA_MASTER_POWDER".UNIT_01.FEEDER_1.LINE_2.POWDER_FLOW)
   END_RUNG
   // the same network as SCL:
   IF "M_ONE" THEN
       "DB16721_POWDER_FLOW_DATA_SAVE_U01_PF1_L2"(iMEDICOAT_DATA := "U01_OERLIKON_1_LINE_2_MEDICOAT_FLOW_CONTROL",   // "FB16700_POWDER_FLOW_DATA_SAVE"
                               ARRAY_NUMBER_MEMORY := "DB16721_POWDER_FLOW_DATA_SAVE_U01_PF1_L2".ARRAY_NUMBER_MEMORY,
                               oMEDICOAT_DATA_ARRAY => "DB16702_OPC_UA_MASTER_POWDER".UNIT_01.FEEDER_1.LINE_2.POWDER_FLOW);
   END_IF;
END_REGION

REGION Network 18: POWDER FEEDER 1 UNIT 01 LINE 2 STATUS
   RUNG wire#powerrail
      Contact( "DB21013_PF_1_HOPPERS_UNIT_01".DATA.FEEDBACK_ON_LINE_2 )
      Coil( "DB16702_OPC_UA_MASTER_POWDER".UNIT_01.FEEDER_1.LINE_2.STATUS.RUNNING )
   END_RUNG
   // the same network as SCL:
   "DB16702_OPC_UA_MASTER_POWDER".UNIT_01.FEEDER_1.LINE_2.STATUS.RUNNING := "DB21013_PF_1_HOPPERS_UNIT_01".DATA.FEEDBACK_ON_LINE_2;
END_REGION

REGION Network 19: POWDER FEEDER 1 UNIT 01 WEIGHT
   RUNG wire#powerrail
      Contact( "M_ONE" )
      Move(in := "DB22150_WP321_WEIGHT_CELLS".WP321DR[0].DR30.GROSS_NET_WEIGHT_X10, out1 => "DB16702_OPC_UA_MASTER_POWDER".UNIT_01.FEEDER_1.WEIGHT)
   END_RUNG
   // the same network as SCL:
   IF "M_ONE" THEN
       "DB16702_OPC_UA_MASTER_POWDER".UNIT_01.FEEDER_1.WEIGHT := "DB22150_WP321_WEIGHT_CELLS".WP321DR[0].DR30.GROSS_NET_WEIGHT_X10;
   END_IF;
END_REGION

REGION Network 20: <<<<<<<<<<<<<< UNIT 02 >>>>>>>>>>>>>>>>>>>>
END_REGION

REGION Network 21: POWDER FEEDER 1 UNIT 02 LINE 1 HOPPER
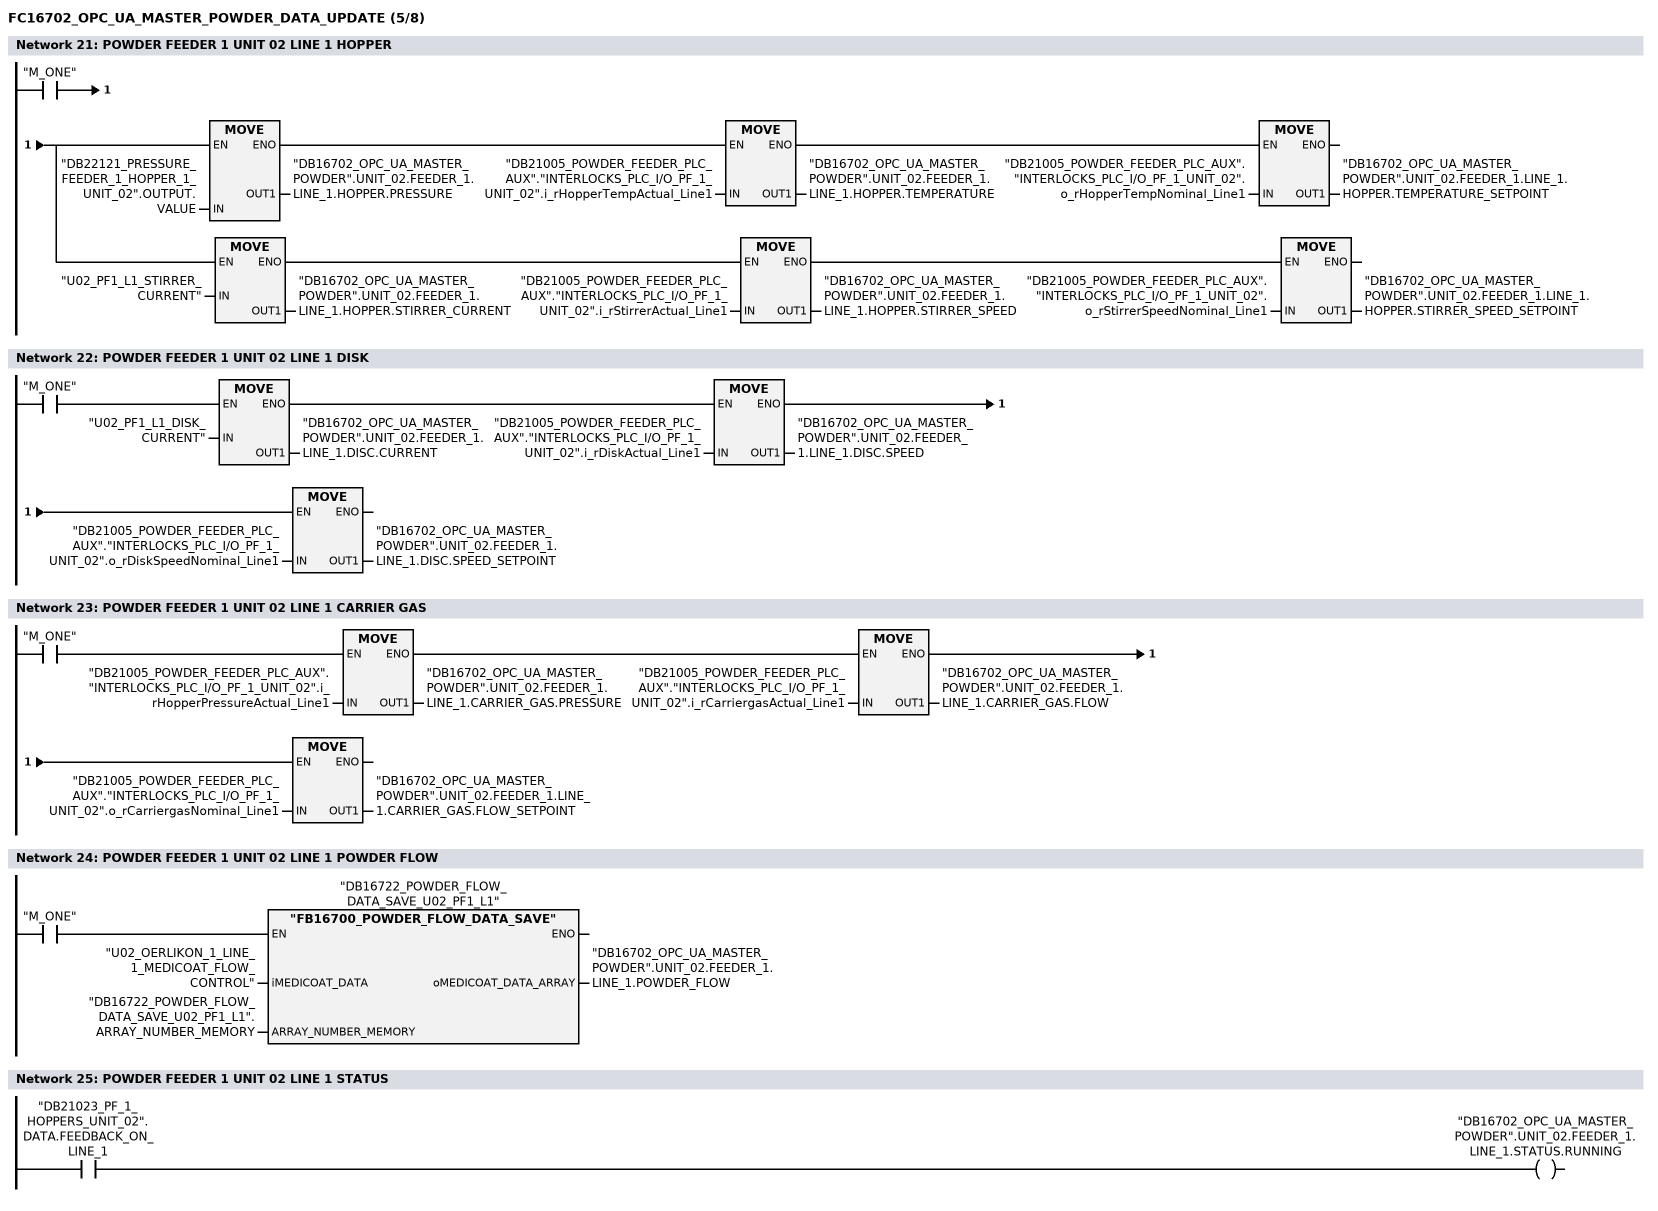
   RUNG wire#powerrail
      Contact( "M_ONE" )
      wire#w1
      Move(in := "DB22121_PRESSURE_FEEDER_1_HOPPER_1_UNIT_02".OUTPUT.VALUE, out1 => "DB16702_OPC_UA_MASTER_POWDER".UNIT_02.FEEDER_1.LINE_1.HOPPER.PRESSURE)
      Move(in := "DB21005_POWDER_FEEDER_PLC_AUX"."INTERLOCKS_PLC_I/O_PF_1_UNIT_02".i_rHopperTempActual_Line1, out1 => "DB16702_OPC_UA_MASTER_POWDER".UNIT_02.FEEDER_1.LINE_1.HOPPER.TEMPERATURE)
      Move(in := "DB21005_POWDER_FEEDER_PLC_AUX"."INTERLOCKS_PLC_I/O_PF_1_UNIT_02".o_rHopperTempNominal_Line1, out1 => "DB16702_OPC_UA_MASTER_POWDER".UNIT_02.FEEDER_1.LINE_1.HOPPER.TEMPERATURE_SETPOINT)
   END_RUNG
   RUNG wire#w1
      Move(in := "U02_PF1_L1_STIRRER_CURRENT", out1 => "DB16702_OPC_UA_MASTER_POWDER".UNIT_02.FEEDER_1.LINE_1.HOPPER.STIRRER_CURRENT)
      Move(in := "DB21005_POWDER_FEEDER_PLC_AUX"."INTERLOCKS_PLC_I/O_PF_1_UNIT_02".i_rStirrerActual_Line1, out1 => "DB16702_OPC_UA_MASTER_POWDER".UNIT_02.FEEDER_1.LINE_1.HOPPER.STIRRER_SPEED)
      Move(in := "DB21005_POWDER_FEEDER_PLC_AUX"."INTERLOCKS_PLC_I/O_PF_1_UNIT_02".o_rStirrerSpeedNominal_Line1, out1 => "DB16702_OPC_UA_MASTER_POWDER".UNIT_02.FEEDER_1.LINE_1.HOPPER.STIRRER_SPEED_SETPOINT)
   END_RUNG
   // the same network as SCL:
   IF "M_ONE" THEN
       "DB16702_OPC_UA_MASTER_POWDER".UNIT_02.FEEDER_1.LINE_1.HOPPER.PRESSURE := "DB22121_PRESSURE_FEEDER_1_HOPPER_1_UNIT_02".OUTPUT.VALUE;
       "DB16702_OPC_UA_MASTER_POWDER".UNIT_02.FEEDER_1.LINE_1.HOPPER.TEMPERATURE := "DB21005_POWDER_FEEDER_PLC_AUX"."INTERLOCKS_PLC_I/O_PF_1_UNIT_02".i_rHopperTempActual_Line1;
       "DB16702_OPC_UA_MASTER_POWDER".UNIT_02.FEEDER_1.LINE_1.HOPPER.TEMPERATURE_SETPOINT := "DB21005_POWDER_FEEDER_PLC_AUX"."INTERLOCKS_PLC_I/O_PF_1_UNIT_02".o_rHopperTempNominal_Line1;
       "DB16702_OPC_UA_MASTER_POWDER".UNIT_02.FEEDER_1.LINE_1.HOPPER.STIRRER_CURRENT := "U02_PF1_L1_STIRRER_CURRENT";
       "DB16702_OPC_UA_MASTER_POWDER".UNIT_02.FEEDER_1.LINE_1.HOPPER.STIRRER_SPEED := "DB21005_POWDER_FEEDER_PLC_AUX"."INTERLOCKS_PLC_I/O_PF_1_UNIT_02".i_rStirrerActual_Line1;
       "DB16702_OPC_UA_MASTER_POWDER".UNIT_02.FEEDER_1.LINE_1.HOPPER.STIRRER_SPEED_SETPOINT := "DB21005_POWDER_FEEDER_PLC_AUX"."INTERLOCKS_PLC_I/O_PF_1_UNIT_02".o_rStirrerSpeedNominal_Line1;
   END_IF;
END_REGION

REGION Network 22: POWDER FEEDER 1 UNIT 02 LINE 1 DISK
   RUNG wire#powerrail
      Contact( "M_ONE" )
      Move(in := "U02_PF1_L1_DISK_CURRENT", out1 => "DB16702_OPC_UA_MASTER_POWDER".UNIT_02.FEEDER_1.LINE_1.DISC.CURRENT)
      Move(in := "DB21005_POWDER_FEEDER_PLC_AUX"."INTERLOCKS_PLC_I/O_PF_1_UNIT_02".i_rDiskActual_Line1, out1 => "DB16702_OPC_UA_MASTER_POWDER".UNIT_02.FEEDER_1.LINE_1.DISC.SPEED)
      Move(in := "DB21005_POWDER_FEEDER_PLC_AUX"."INTERLOCKS_PLC_I/O_PF_1_UNIT_02".o_rDiskSpeedNominal_Line1, out1 => "DB16702_OPC_UA_MASTER_POWDER".UNIT_02.FEEDER_1.LINE_1.DISC.SPEED_SETPOINT)
   END_RUNG
   // the same network as SCL:
   IF "M_ONE" THEN
       "DB16702_OPC_UA_MASTER_POWDER".UNIT_02.FEEDER_1.LINE_1.DISC.CURRENT := "U02_PF1_L1_DISK_CURRENT";
       "DB16702_OPC_UA_MASTER_POWDER".UNIT_02.FEEDER_1.LINE_1.DISC.SPEED := "DB21005_POWDER_FEEDER_PLC_AUX"."INTERLOCKS_PLC_I/O_PF_1_UNIT_02".i_rDiskActual_Line1;
       "DB16702_OPC_UA_MASTER_POWDER".UNIT_02.FEEDER_1.LINE_1.DISC.SPEED_SETPOINT := "DB21005_POWDER_FEEDER_PLC_AUX"."INTERLOCKS_PLC_I/O_PF_1_UNIT_02".o_rDiskSpeedNominal_Line1;
   END_IF;
END_REGION

REGION Network 23: POWDER FEEDER 1 UNIT 02 LINE 1 CARRIER GAS
   RUNG wire#powerrail
      Contact( "M_ONE" )
      Move(in := "DB21005_POWDER_FEEDER_PLC_AUX"."INTERLOCKS_PLC_I/O_PF_1_UNIT_02".i_rHopperPressureActual_Line1, out1 => "DB16702_OPC_UA_MASTER_POWDER".UNIT_02.FEEDER_1.LINE_1.CARRIER_GAS.PRESSURE)
      Move(in := "DB21005_POWDER_FEEDER_PLC_AUX"."INTERLOCKS_PLC_I/O_PF_1_UNIT_02".i_rCarriergasActual_Line1, out1 => "DB16702_OPC_UA_MASTER_POWDER".UNIT_02.FEEDER_1.LINE_1.CARRIER_GAS.FLOW)
      Move(in := "DB21005_POWDER_FEEDER_PLC_AUX"."INTERLOCKS_PLC_I/O_PF_1_UNIT_02".o_rCarriergasNominal_Line1, out1 => "DB16702_OPC_UA_MASTER_POWDER".UNIT_02.FEEDER_1.LINE_1.CARRIER_GAS.FLOW_SETPOINT)
   END_RUNG
   // the same network as SCL:
   IF "M_ONE" THEN
       "DB16702_OPC_UA_MASTER_POWDER".UNIT_02.FEEDER_1.LINE_1.CARRIER_GAS.PRESSURE := "DB21005_POWDER_FEEDER_PLC_AUX"."INTERLOCKS_PLC_I/O_PF_1_UNIT_02".i_rHopperPressureActual_Line1;
       "DB16702_OPC_UA_MASTER_POWDER".UNIT_02.FEEDER_1.LINE_1.CARRIER_GAS.FLOW := "DB21005_POWDER_FEEDER_PLC_AUX"."INTERLOCKS_PLC_I/O_PF_1_UNIT_02".i_rCarriergasActual_Line1;
       "DB16702_OPC_UA_MASTER_POWDER".UNIT_02.FEEDER_1.LINE_1.CARRIER_GAS.FLOW_SETPOINT := "DB21005_POWDER_FEEDER_PLC_AUX"."INTERLOCKS_PLC_I/O_PF_1_UNIT_02".o_rCarriergasNominal_Line1;
   END_IF;
END_REGION

REGION Network 24: POWDER FEEDER 1 UNIT 02 LINE 1 POWDER FLOW
   RUNG wire#powerrail
      Contact( "M_ONE" )
      "DB16722_POWDER_FLOW_DATA_SAVE_U02_PF1_L1"(iMEDICOAT_DATA := "U02_OERLIKON_1_LINE_1_MEDICOAT_FLOW_CONTROL", ARRAY_NUMBER_MEMORY := "DB16722_POWDER_FLOW_DATA_SAVE_U02_PF1_L1".ARRAY_NUMBER_MEMORY, oMEDICOAT_DATA_ARRAY => "DB16702_OPC_UA_MASTER_POWDER".UNIT_02.FEEDER_1.LINE_1.POWDER_FLOW)
   END_RUNG
   // the same network as SCL:
   IF "M_ONE" THEN
       "DB16722_POWDER_FLOW_DATA_SAVE_U02_PF1_L1"(iMEDICOAT_DATA := "U02_OERLIKON_1_LINE_1_MEDICOAT_FLOW_CONTROL",   // "FB16700_POWDER_FLOW_DATA_SAVE"
                               ARRAY_NUMBER_MEMORY := "DB16722_POWDER_FLOW_DATA_SAVE_U02_PF1_L1".ARRAY_NUMBER_MEMORY,
                               oMEDICOAT_DATA_ARRAY => "DB16702_OPC_UA_MASTER_POWDER".UNIT_02.FEEDER_1.LINE_1.POWDER_FLOW);
   END_IF;
END_REGION

REGION Network 25: POWDER FEEDER 1 UNIT 02 LINE 1 STATUS
   RUNG wire#powerrail
      Contact( "DB21023_PF_1_HOPPERS_UNIT_02".DATA.FEEDBACK_ON_LINE_1 )
      Coil( "DB16702_OPC_UA_MASTER_POWDER".UNIT_02.FEEDER_1.LINE_1.STATUS.RUNNING )
   END_RUNG
   // the same network as SCL:
   "DB16702_OPC_UA_MASTER_POWDER".UNIT_02.FEEDER_1.LINE_1.STATUS.RUNNING := "DB21023_PF_1_HOPPERS_UNIT_02".DATA.FEEDBACK_ON_LINE_1;
END_REGION

REGION Network 26: POWDER FEEDER 1 UNIT 02 LINE 2 HOPPER
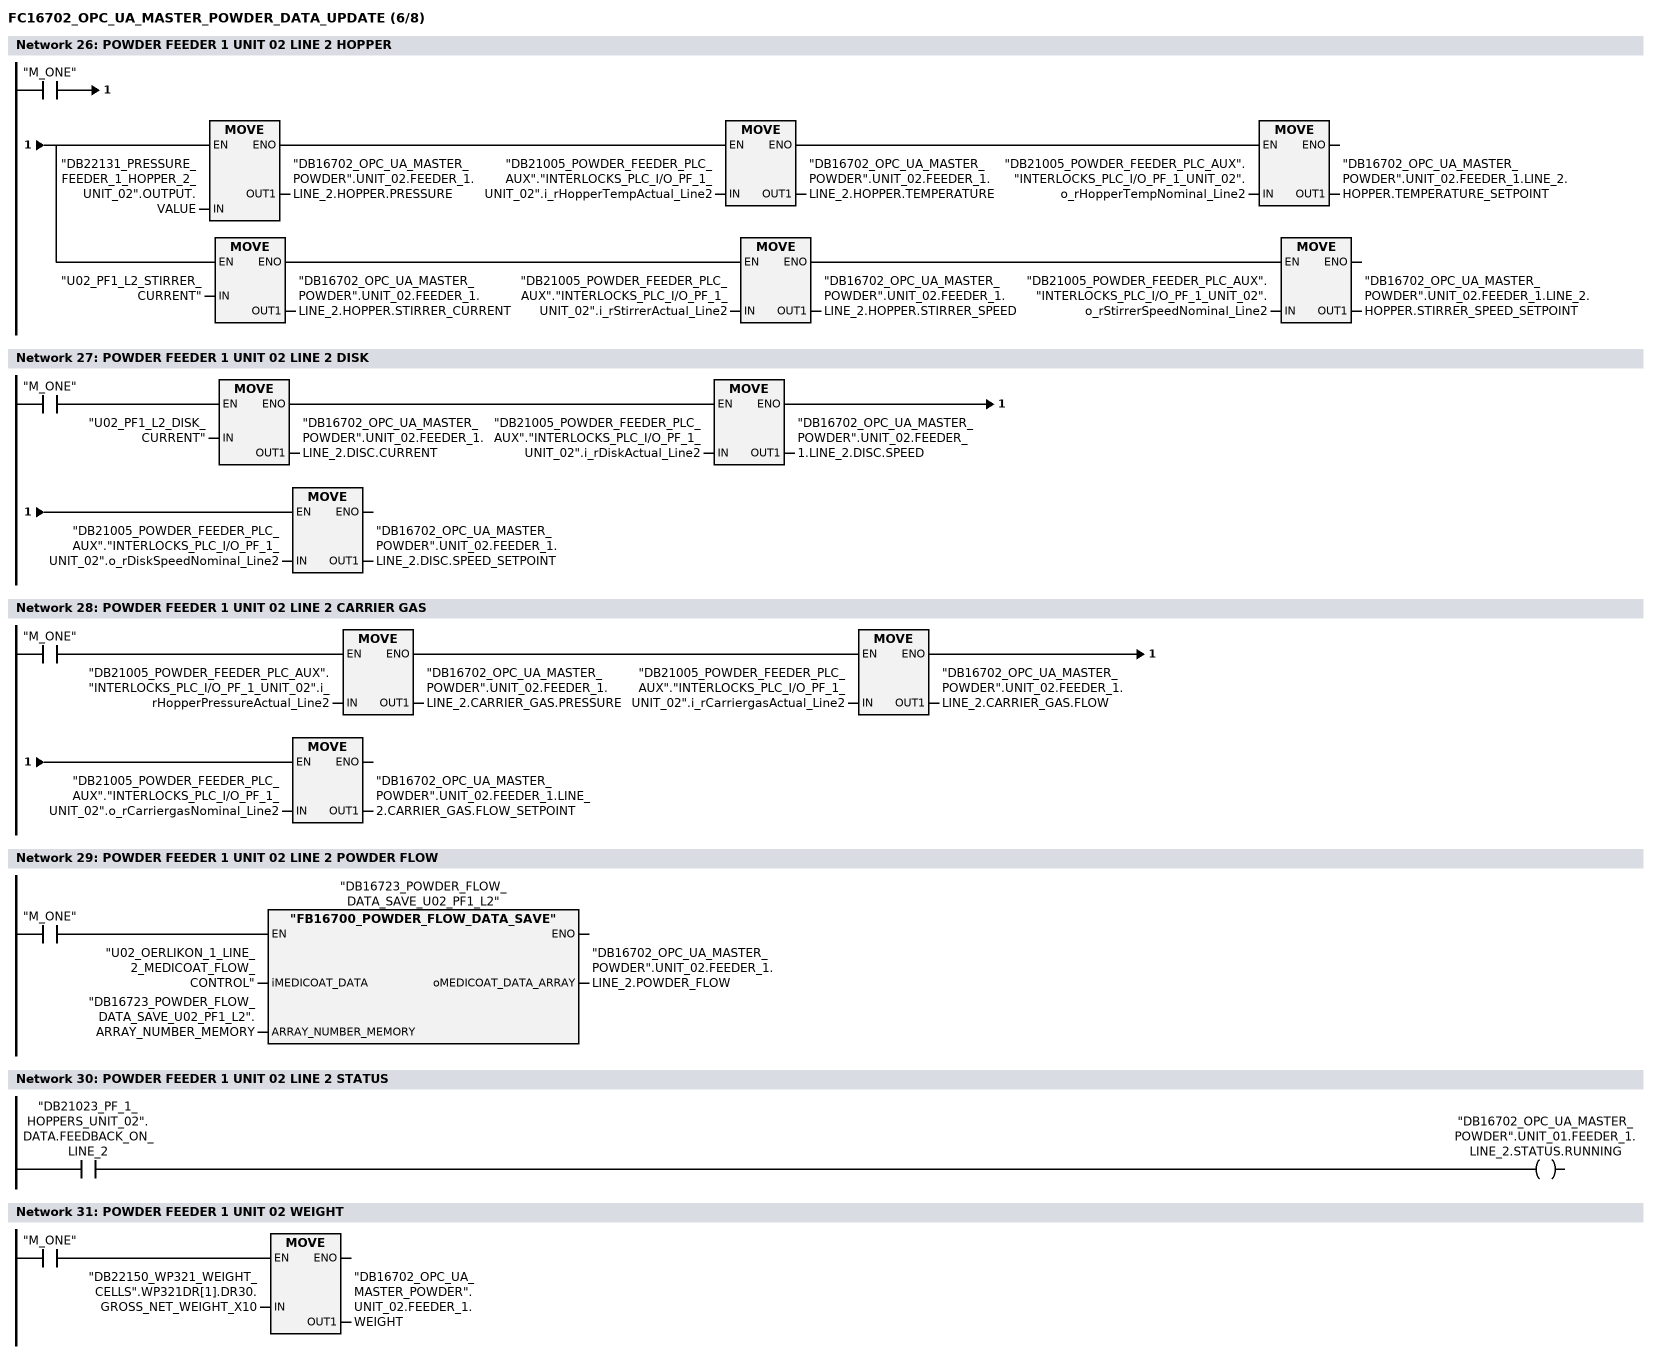
   RUNG wire#powerrail
      Contact( "M_ONE" )
      wire#w1
      Move(in := "DB22131_PRESSURE_FEEDER_1_HOPPER_2_UNIT_02".OUTPUT.VALUE, out1 => "DB16702_OPC_UA_MASTER_POWDER".UNIT_02.FEEDER_1.LINE_2.HOPPER.PRESSURE)
      Move(in := "DB21005_POWDER_FEEDER_PLC_AUX"."INTERLOCKS_PLC_I/O_PF_1_UNIT_02".i_rHopperTempActual_Line2, out1 => "DB16702_OPC_UA_MASTER_POWDER".UNIT_02.FEEDER_1.LINE_2.HOPPER.TEMPERATURE)
      Move(in := "DB21005_POWDER_FEEDER_PLC_AUX"."INTERLOCKS_PLC_I/O_PF_1_UNIT_02".o_rHopperTempNominal_Line2, out1 => "DB16702_OPC_UA_MASTER_POWDER".UNIT_02.FEEDER_1.LINE_2.HOPPER.TEMPERATURE_SETPOINT)
   END_RUNG
   RUNG wire#w1
      Move(in := "U02_PF1_L2_STIRRER_CURRENT", out1 => "DB16702_OPC_UA_MASTER_POWDER".UNIT_02.FEEDER_1.LINE_2.HOPPER.STIRRER_CURRENT)
      Move(in := "DB21005_POWDER_FEEDER_PLC_AUX"."INTERLOCKS_PLC_I/O_PF_1_UNIT_02".i_rStirrerActual_Line2, out1 => "DB16702_OPC_UA_MASTER_POWDER".UNIT_02.FEEDER_1.LINE_2.HOPPER.STIRRER_SPEED)
      Move(in := "DB21005_POWDER_FEEDER_PLC_AUX"."INTERLOCKS_PLC_I/O_PF_1_UNIT_02".o_rStirrerSpeedNominal_Line2, out1 => "DB16702_OPC_UA_MASTER_POWDER".UNIT_02.FEEDER_1.LINE_2.HOPPER.STIRRER_SPEED_SETPOINT)
   END_RUNG
   // the same network as SCL:
   IF "M_ONE" THEN
       "DB16702_OPC_UA_MASTER_POWDER".UNIT_02.FEEDER_1.LINE_2.HOPPER.PRESSURE := "DB22131_PRESSURE_FEEDER_1_HOPPER_2_UNIT_02".OUTPUT.VALUE;
       "DB16702_OPC_UA_MASTER_POWDER".UNIT_02.FEEDER_1.LINE_2.HOPPER.TEMPERATURE := "DB21005_POWDER_FEEDER_PLC_AUX"."INTERLOCKS_PLC_I/O_PF_1_UNIT_02".i_rHopperTempActual_Line2;
       "DB16702_OPC_UA_MASTER_POWDER".UNIT_02.FEEDER_1.LINE_2.HOPPER.TEMPERATURE_SETPOINT := "DB21005_POWDER_FEEDER_PLC_AUX"."INTERLOCKS_PLC_I/O_PF_1_UNIT_02".o_rHopperTempNominal_Line2;
       "DB16702_OPC_UA_MASTER_POWDER".UNIT_02.FEEDER_1.LINE_2.HOPPER.STIRRER_CURRENT := "U02_PF1_L2_STIRRER_CURRENT";
       "DB16702_OPC_UA_MASTER_POWDER".UNIT_02.FEEDER_1.LINE_2.HOPPER.STIRRER_SPEED := "DB21005_POWDER_FEEDER_PLC_AUX"."INTERLOCKS_PLC_I/O_PF_1_UNIT_02".i_rStirrerActual_Line2;
       "DB16702_OPC_UA_MASTER_POWDER".UNIT_02.FEEDER_1.LINE_2.HOPPER.STIRRER_SPEED_SETPOINT := "DB21005_POWDER_FEEDER_PLC_AUX"."INTERLOCKS_PLC_I/O_PF_1_UNIT_02".o_rStirrerSpeedNominal_Line2;
   END_IF;
END_REGION

REGION Network 27: POWDER FEEDER 1 UNIT 02 LINE 2 DISK
   RUNG wire#powerrail
      Contact( "M_ONE" )
      Move(in := "U02_PF1_L2_DISK_CURRENT", out1 => "DB16702_OPC_UA_MASTER_POWDER".UNIT_02.FEEDER_1.LINE_2.DISC.CURRENT)
      Move(in := "DB21005_POWDER_FEEDER_PLC_AUX"."INTERLOCKS_PLC_I/O_PF_1_UNIT_02".i_rDiskActual_Line2, out1 => "DB16702_OPC_UA_MASTER_POWDER".UNIT_02.FEEDER_1.LINE_2.DISC.SPEED)
      Move(in := "DB21005_POWDER_FEEDER_PLC_AUX"."INTERLOCKS_PLC_I/O_PF_1_UNIT_02".o_rDiskSpeedNominal_Line2, out1 => "DB16702_OPC_UA_MASTER_POWDER".UNIT_02.FEEDER_1.LINE_2.DISC.SPEED_SETPOINT)
   END_RUNG
   // the same network as SCL:
   IF "M_ONE" THEN
       "DB16702_OPC_UA_MASTER_POWDER".UNIT_02.FEEDER_1.LINE_2.DISC.CURRENT := "U02_PF1_L2_DISK_CURRENT";
       "DB16702_OPC_UA_MASTER_POWDER".UNIT_02.FEEDER_1.LINE_2.DISC.SPEED := "DB21005_POWDER_FEEDER_PLC_AUX"."INTERLOCKS_PLC_I/O_PF_1_UNIT_02".i_rDiskActual_Line2;
       "DB16702_OPC_UA_MASTER_POWDER".UNIT_02.FEEDER_1.LINE_2.DISC.SPEED_SETPOINT := "DB21005_POWDER_FEEDER_PLC_AUX"."INTERLOCKS_PLC_I/O_PF_1_UNIT_02".o_rDiskSpeedNominal_Line2;
   END_IF;
END_REGION

REGION Network 28: POWDER FEEDER 1 UNIT 02 LINE 2 CARRIER GAS
   RUNG wire#powerrail
      Contact( "M_ONE" )
      Move(in := "DB21005_POWDER_FEEDER_PLC_AUX"."INTERLOCKS_PLC_I/O_PF_1_UNIT_02".i_rHopperPressureActual_Line2, out1 => "DB16702_OPC_UA_MASTER_POWDER".UNIT_02.FEEDER_1.LINE_2.CARRIER_GAS.PRESSURE)
      Move(in := "DB21005_POWDER_FEEDER_PLC_AUX"."INTERLOCKS_PLC_I/O_PF_1_UNIT_02".i_rCarriergasActual_Line2, out1 => "DB16702_OPC_UA_MASTER_POWDER".UNIT_02.FEEDER_1.LINE_2.CARRIER_GAS.FLOW)
      Move(in := "DB21005_POWDER_FEEDER_PLC_AUX"."INTERLOCKS_PLC_I/O_PF_1_UNIT_02".o_rCarriergasNominal_Line2, out1 => "DB16702_OPC_UA_MASTER_POWDER".UNIT_02.FEEDER_1.LINE_2.CARRIER_GAS.FLOW_SETPOINT)
   END_RUNG
   // the same network as SCL:
   IF "M_ONE" THEN
       "DB16702_OPC_UA_MASTER_POWDER".UNIT_02.FEEDER_1.LINE_2.CARRIER_GAS.PRESSURE := "DB21005_POWDER_FEEDER_PLC_AUX"."INTERLOCKS_PLC_I/O_PF_1_UNIT_02".i_rHopperPressureActual_Line2;
       "DB16702_OPC_UA_MASTER_POWDER".UNIT_02.FEEDER_1.LINE_2.CARRIER_GAS.FLOW := "DB21005_POWDER_FEEDER_PLC_AUX"."INTERLOCKS_PLC_I/O_PF_1_UNIT_02".i_rCarriergasActual_Line2;
       "DB16702_OPC_UA_MASTER_POWDER".UNIT_02.FEEDER_1.LINE_2.CARRIER_GAS.FLOW_SETPOINT := "DB21005_POWDER_FEEDER_PLC_AUX"."INTERLOCKS_PLC_I/O_PF_1_UNIT_02".o_rCarriergasNominal_Line2;
   END_IF;
END_REGION

REGION Network 29: POWDER FEEDER 1 UNIT 02 LINE 2 POWDER FLOW
   RUNG wire#powerrail
      Contact( "M_ONE" )
      "DB16723_POWDER_FLOW_DATA_SAVE_U02_PF1_L2"(iMEDICOAT_DATA := "U02_OERLIKON_1_LINE_2_MEDICOAT_FLOW_CONTROL", ARRAY_NUMBER_MEMORY := "DB16723_POWDER_FLOW_DATA_SAVE_U02_PF1_L2".ARRAY_NUMBER_MEMORY, oMEDICOAT_DATA_ARRAY => "DB16702_OPC_UA_MASTER_POWDER".UNIT_02.FEEDER_1.LINE_2.POWDER_FLOW)
   END_RUNG
   // the same network as SCL:
   IF "M_ONE" THEN
       "DB16723_POWDER_FLOW_DATA_SAVE_U02_PF1_L2"(iMEDICOAT_DATA := "U02_OERLIKON_1_LINE_2_MEDICOAT_FLOW_CONTROL",   // "FB16700_POWDER_FLOW_DATA_SAVE"
                               ARRAY_NUMBER_MEMORY := "DB16723_POWDER_FLOW_DATA_SAVE_U02_PF1_L2".ARRAY_NUMBER_MEMORY,
                               oMEDICOAT_DATA_ARRAY => "DB16702_OPC_UA_MASTER_POWDER".UNIT_02.FEEDER_1.LINE_2.POWDER_FLOW);
   END_IF;
END_REGION

REGION Network 30: POWDER FEEDER 1 UNIT 02 LINE 2 STATUS
   RUNG wire#powerrail
      Contact( "DB21023_PF_1_HOPPERS_UNIT_02".DATA.FEEDBACK_ON_LINE_2 )
      Coil( "DB16702_OPC_UA_MASTER_POWDER".UNIT_01.FEEDER_1.LINE_2.STATUS.RUNNING )
   END_RUNG
   // the same network as SCL:
   "DB16702_OPC_UA_MASTER_POWDER".UNIT_01.FEEDER_1.LINE_2.STATUS.RUNNING := "DB21023_PF_1_HOPPERS_UNIT_02".DATA.FEEDBACK_ON_LINE_2;
END_REGION

REGION Network 31: POWDER FEEDER 1 UNIT 02 WEIGHT
   RUNG wire#powerrail
      Contact( "M_ONE" )
      Move(in := "DB22150_WP321_WEIGHT_CELLS".WP321DR[1].DR30.GROSS_NET_WEIGHT_X10, out1 => "DB16702_OPC_UA_MASTER_POWDER".UNIT_02.FEEDER_1.WEIGHT)
   END_RUNG
   // the same network as SCL:
   IF "M_ONE" THEN
       "DB16702_OPC_UA_MASTER_POWDER".UNIT_02.FEEDER_1.WEIGHT := "DB22150_WP321_WEIGHT_CELLS".WP321DR[1].DR30.GROSS_NET_WEIGHT_X10;
   END_IF;
END_REGION

REGION Network 32: POWDER FEEDER 2 UNIT 02 LINE 1 HOPPER
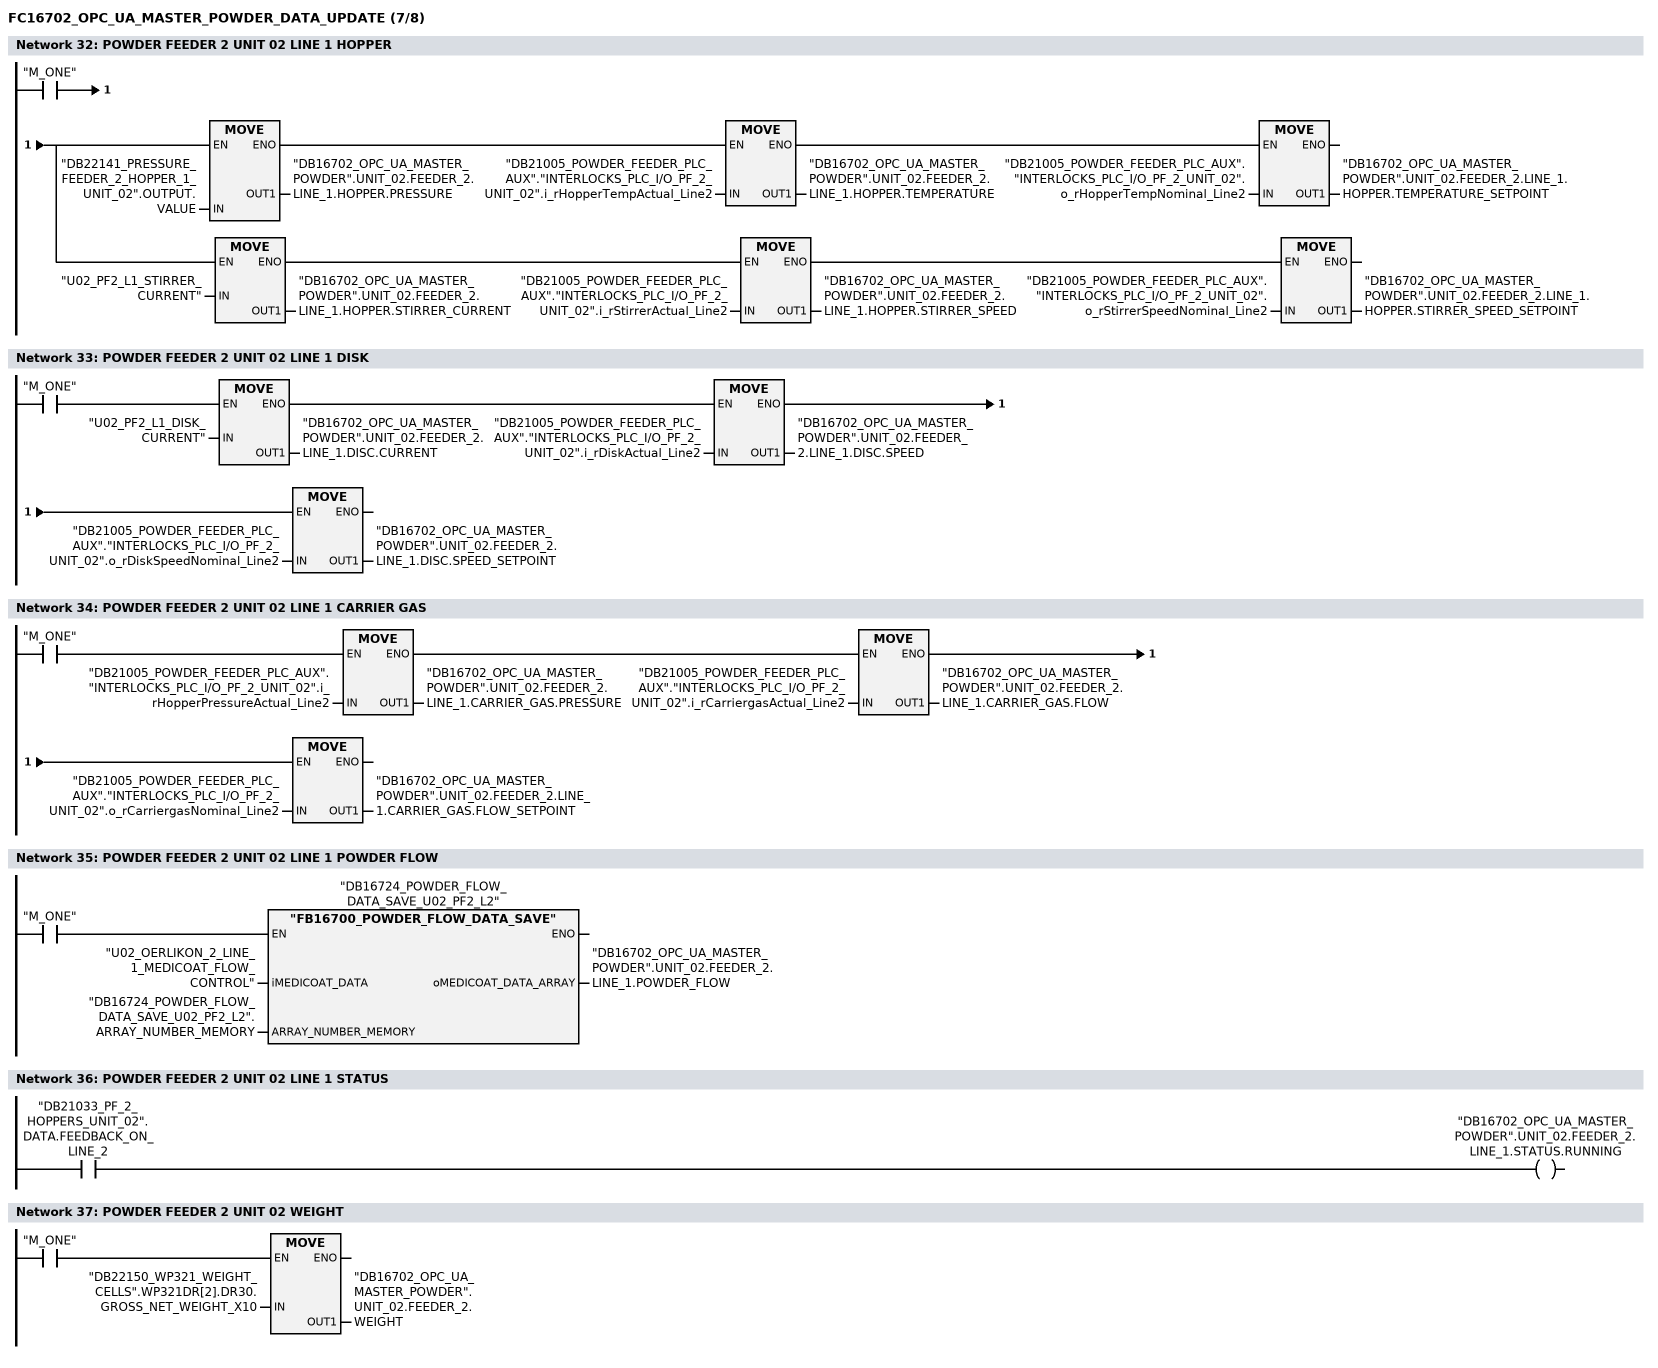
   RUNG wire#powerrail
      Contact( "M_ONE" )
      wire#w1
      Move(in := "DB22141_PRESSURE_FEEDER_2_HOPPER_1_UNIT_02".OUTPUT.VALUE, out1 => "DB16702_OPC_UA_MASTER_POWDER".UNIT_02.FEEDER_2.LINE_1.HOPPER.PRESSURE)
      Move(in := "DB21005_POWDER_FEEDER_PLC_AUX"."INTERLOCKS_PLC_I/O_PF_2_UNIT_02".i_rHopperTempActual_Line2, out1 => "DB16702_OPC_UA_MASTER_POWDER".UNIT_02.FEEDER_2.LINE_1.HOPPER.TEMPERATURE)
      Move(in := "DB21005_POWDER_FEEDER_PLC_AUX"."INTERLOCKS_PLC_I/O_PF_2_UNIT_02".o_rHopperTempNominal_Line2, out1 => "DB16702_OPC_UA_MASTER_POWDER".UNIT_02.FEEDER_2.LINE_1.HOPPER.TEMPERATURE_SETPOINT)
   END_RUNG
   RUNG wire#w1
      Move(in := "U02_PF2_L1_STIRRER_CURRENT", out1 => "DB16702_OPC_UA_MASTER_POWDER".UNIT_02.FEEDER_2.LINE_1.HOPPER.STIRRER_CURRENT)
      Move(in := "DB21005_POWDER_FEEDER_PLC_AUX"."INTERLOCKS_PLC_I/O_PF_2_UNIT_02".i_rStirrerActual_Line2, out1 => "DB16702_OPC_UA_MASTER_POWDER".UNIT_02.FEEDER_2.LINE_1.HOPPER.STIRRER_SPEED)
      Move(in := "DB21005_POWDER_FEEDER_PLC_AUX"."INTERLOCKS_PLC_I/O_PF_2_UNIT_02".o_rStirrerSpeedNominal_Line2, out1 => "DB16702_OPC_UA_MASTER_POWDER".UNIT_02.FEEDER_2.LINE_1.HOPPER.STIRRER_SPEED_SETPOINT)
   END_RUNG
   // the same network as SCL:
   IF "M_ONE" THEN
       "DB16702_OPC_UA_MASTER_POWDER".UNIT_02.FEEDER_2.LINE_1.HOPPER.PRESSURE := "DB22141_PRESSURE_FEEDER_2_HOPPER_1_UNIT_02".OUTPUT.VALUE;
       "DB16702_OPC_UA_MASTER_POWDER".UNIT_02.FEEDER_2.LINE_1.HOPPER.TEMPERATURE := "DB21005_POWDER_FEEDER_PLC_AUX"."INTERLOCKS_PLC_I/O_PF_2_UNIT_02".i_rHopperTempActual_Line2;
       "DB16702_OPC_UA_MASTER_POWDER".UNIT_02.FEEDER_2.LINE_1.HOPPER.TEMPERATURE_SETPOINT := "DB21005_POWDER_FEEDER_PLC_AUX"."INTERLOCKS_PLC_I/O_PF_2_UNIT_02".o_rHopperTempNominal_Line2;
       "DB16702_OPC_UA_MASTER_POWDER".UNIT_02.FEEDER_2.LINE_1.HOPPER.STIRRER_CURRENT := "U02_PF2_L1_STIRRER_CURRENT";
       "DB16702_OPC_UA_MASTER_POWDER".UNIT_02.FEEDER_2.LINE_1.HOPPER.STIRRER_SPEED := "DB21005_POWDER_FEEDER_PLC_AUX"."INTERLOCKS_PLC_I/O_PF_2_UNIT_02".i_rStirrerActual_Line2;
       "DB16702_OPC_UA_MASTER_POWDER".UNIT_02.FEEDER_2.LINE_1.HOPPER.STIRRER_SPEED_SETPOINT := "DB21005_POWDER_FEEDER_PLC_AUX"."INTERLOCKS_PLC_I/O_PF_2_UNIT_02".o_rStirrerSpeedNominal_Line2;
   END_IF;
END_REGION

REGION Network 33: POWDER FEEDER 2 UNIT 02 LINE 1 DISK
   RUNG wire#powerrail
      Contact( "M_ONE" )
      Move(in := "U02_PF2_L1_DISK_CURRENT", out1 => "DB16702_OPC_UA_MASTER_POWDER".UNIT_02.FEEDER_2.LINE_1.DISC.CURRENT)
      Move(in := "DB21005_POWDER_FEEDER_PLC_AUX"."INTERLOCKS_PLC_I/O_PF_2_UNIT_02".i_rDiskActual_Line2, out1 => "DB16702_OPC_UA_MASTER_POWDER".UNIT_02.FEEDER_2.LINE_1.DISC.SPEED)
      Move(in := "DB21005_POWDER_FEEDER_PLC_AUX"."INTERLOCKS_PLC_I/O_PF_2_UNIT_02".o_rDiskSpeedNominal_Line2, out1 => "DB16702_OPC_UA_MASTER_POWDER".UNIT_02.FEEDER_2.LINE_1.DISC.SPEED_SETPOINT)
   END_RUNG
   // the same network as SCL:
   IF "M_ONE" THEN
       "DB16702_OPC_UA_MASTER_POWDER".UNIT_02.FEEDER_2.LINE_1.DISC.CURRENT := "U02_PF2_L1_DISK_CURRENT";
       "DB16702_OPC_UA_MASTER_POWDER".UNIT_02.FEEDER_2.LINE_1.DISC.SPEED := "DB21005_POWDER_FEEDER_PLC_AUX"."INTERLOCKS_PLC_I/O_PF_2_UNIT_02".i_rDiskActual_Line2;
       "DB16702_OPC_UA_MASTER_POWDER".UNIT_02.FEEDER_2.LINE_1.DISC.SPEED_SETPOINT := "DB21005_POWDER_FEEDER_PLC_AUX"."INTERLOCKS_PLC_I/O_PF_2_UNIT_02".o_rDiskSpeedNominal_Line2;
   END_IF;
END_REGION

REGION Network 34: POWDER FEEDER 2 UNIT 02 LINE 1 CARRIER GAS
   RUNG wire#powerrail
      Contact( "M_ONE" )
      Move(in := "DB21005_POWDER_FEEDER_PLC_AUX"."INTERLOCKS_PLC_I/O_PF_2_UNIT_02".i_rHopperPressureActual_Line2, out1 => "DB16702_OPC_UA_MASTER_POWDER".UNIT_02.FEEDER_2.LINE_1.CARRIER_GAS.PRESSURE)
      Move(in := "DB21005_POWDER_FEEDER_PLC_AUX"."INTERLOCKS_PLC_I/O_PF_2_UNIT_02".i_rCarriergasActual_Line2, out1 => "DB16702_OPC_UA_MASTER_POWDER".UNIT_02.FEEDER_2.LINE_1.CARRIER_GAS.FLOW)
      Move(in := "DB21005_POWDER_FEEDER_PLC_AUX"."INTERLOCKS_PLC_I/O_PF_2_UNIT_02".o_rCarriergasNominal_Line2, out1 => "DB16702_OPC_UA_MASTER_POWDER".UNIT_02.FEEDER_2.LINE_1.CARRIER_GAS.FLOW_SETPOINT)
   END_RUNG
   // the same network as SCL:
   IF "M_ONE" THEN
       "DB16702_OPC_UA_MASTER_POWDER".UNIT_02.FEEDER_2.LINE_1.CARRIER_GAS.PRESSURE := "DB21005_POWDER_FEEDER_PLC_AUX"."INTERLOCKS_PLC_I/O_PF_2_UNIT_02".i_rHopperPressureActual_Line2;
       "DB16702_OPC_UA_MASTER_POWDER".UNIT_02.FEEDER_2.LINE_1.CARRIER_GAS.FLOW := "DB21005_POWDER_FEEDER_PLC_AUX"."INTERLOCKS_PLC_I/O_PF_2_UNIT_02".i_rCarriergasActual_Line2;
       "DB16702_OPC_UA_MASTER_POWDER".UNIT_02.FEEDER_2.LINE_1.CARRIER_GAS.FLOW_SETPOINT := "DB21005_POWDER_FEEDER_PLC_AUX"."INTERLOCKS_PLC_I/O_PF_2_UNIT_02".o_rCarriergasNominal_Line2;
   END_IF;
END_REGION

REGION Network 35: POWDER FEEDER 2 UNIT 02 LINE 1 POWDER FLOW
   RUNG wire#powerrail
      Contact( "M_ONE" )
      "DB16724_POWDER_FLOW_DATA_SAVE_U02_PF2_L2"(iMEDICOAT_DATA := "U02_OERLIKON_2_LINE_1_MEDICOAT_FLOW_CONTROL", ARRAY_NUMBER_MEMORY := "DB16724_POWDER_FLOW_DATA_SAVE_U02_PF2_L2".ARRAY_NUMBER_MEMORY, oMEDICOAT_DATA_ARRAY => "DB16702_OPC_UA_MASTER_POWDER".UNIT_02.FEEDER_2.LINE_1.POWDER_FLOW)
   END_RUNG
   // the same network as SCL:
   IF "M_ONE" THEN
       "DB16724_POWDER_FLOW_DATA_SAVE_U02_PF2_L2"(iMEDICOAT_DATA := "U02_OERLIKON_2_LINE_1_MEDICOAT_FLOW_CONTROL",   // "FB16700_POWDER_FLOW_DATA_SAVE"
                               ARRAY_NUMBER_MEMORY := "DB16724_POWDER_FLOW_DATA_SAVE_U02_PF2_L2".ARRAY_NUMBER_MEMORY,
                               oMEDICOAT_DATA_ARRAY => "DB16702_OPC_UA_MASTER_POWDER".UNIT_02.FEEDER_2.LINE_1.POWDER_FLOW);
   END_IF;
END_REGION

REGION Network 36: POWDER FEEDER 2 UNIT 02 LINE 1 STATUS
   RUNG wire#powerrail
      Contact( "DB21033_PF_2_HOPPERS_UNIT_02".DATA.FEEDBACK_ON_LINE_2 )
      Coil( "DB16702_OPC_UA_MASTER_POWDER".UNIT_02.FEEDER_2.LINE_1.STATUS.RUNNING )
   END_RUNG
   // the same network as SCL:
   "DB16702_OPC_UA_MASTER_POWDER".UNIT_02.FEEDER_2.LINE_1.STATUS.RUNNING := "DB21033_PF_2_HOPPERS_UNIT_02".DATA.FEEDBACK_ON_LINE_2;
END_REGION

REGION Network 37: POWDER FEEDER 2 UNIT 02 WEIGHT
   RUNG wire#powerrail
      Contact( "M_ONE" )
      Move(in := "DB22150_WP321_WEIGHT_CELLS".WP321DR[2].DR30.GROSS_NET_WEIGHT_X10, out1 => "DB16702_OPC_UA_MASTER_POWDER".UNIT_02.FEEDER_2.WEIGHT)
   END_RUNG
   // the same network as SCL:
   IF "M_ONE" THEN
       "DB16702_OPC_UA_MASTER_POWDER".UNIT_02.FEEDER_2.WEIGHT := "DB22150_WP321_WEIGHT_CELLS".WP321DR[2].DR30.GROSS_NET_WEIGHT_X10;
   END_IF;
END_REGION

REGION Network 38: UNIT 02 COMBINER POWDER FLOW
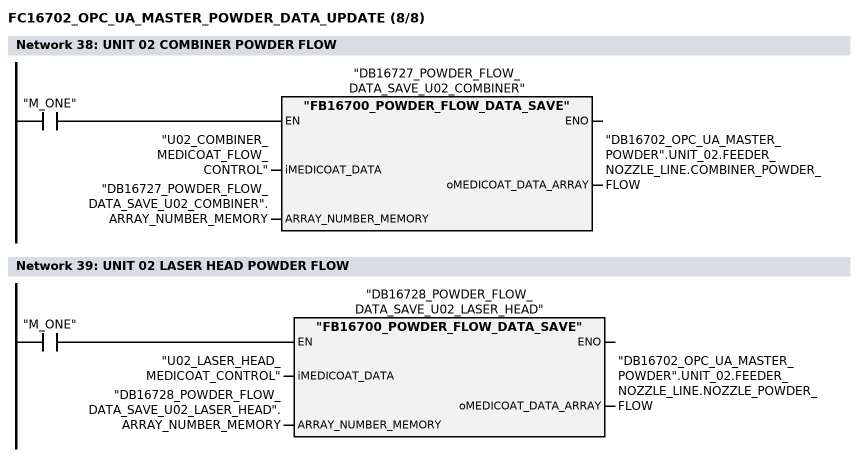
   RUNG wire#powerrail
      Contact( "M_ONE" )
      "DB16727_POWDER_FLOW_DATA_SAVE_U02_COMBINER"(iMEDICOAT_DATA := "U02_COMBINER_MEDICOAT_FLOW_CONTROL", ARRAY_NUMBER_MEMORY := "DB16727_POWDER_FLOW_DATA_SAVE_U02_COMBINER".ARRAY_NUMBER_MEMORY, oMEDICOAT_DATA_ARRAY => "DB16702_OPC_UA_MASTER_POWDER".UNIT_02.FEEDER_NOZZLE_LINE.COMBINER_POWDER_FLOW)
   END_RUNG
   // the same network as SCL:
   IF "M_ONE" THEN
       "DB16727_POWDER_FLOW_DATA_SAVE_U02_COMBINER"(iMEDICOAT_DATA := "U02_COMBINER_MEDICOAT_FLOW_CONTROL",   // "FB16700_POWDER_FLOW_DATA_SAVE"
                               ARRAY_NUMBER_MEMORY := "DB16727_POWDER_FLOW_DATA_SAVE_U02_COMBINER".ARRAY_NUMBER_MEMORY,
                               oMEDICOAT_DATA_ARRAY => "DB16702_OPC_UA_MASTER_POWDER".UNIT_02.FEEDER_NOZZLE_LINE.COMBINER_POWDER_FLOW);
   END_IF;
END_REGION

REGION Network 39: UNIT 02 LASER HEAD POWDER FLOW
   RUNG wire#powerrail
      Contact( "M_ONE" )
      "DB16728_POWDER_FLOW_DATA_SAVE_U02_LASER_HEAD"(iMEDICOAT_DATA := "U02_LASER_HEAD_MEDICOAT_CONTROL", ARRAY_NUMBER_MEMORY := "DB16728_POWDER_FLOW_DATA_SAVE_U02_LASER_HEAD".ARRAY_NUMBER_MEMORY, oMEDICOAT_DATA_ARRAY => "DB16702_OPC_UA_MASTER_POWDER".UNIT_02.FEEDER_NOZZLE_LINE.NOZZLE_POWDER_FLOW)
   END_RUNG
   // the same network as SCL:
   IF "M_ONE" THEN
       "DB16728_POWDER_FLOW_DATA_SAVE_U02_LASER_HEAD"(iMEDICOAT_DATA := "U02_LASER_HEAD_MEDICOAT_CONTROL",   // "FB16700_POWDER_FLOW_DATA_SAVE"
                               ARRAY_NUMBER_MEMORY := "DB16728_POWDER_FLOW_DATA_SAVE_U02_LASER_HEAD".ARRAY_NUMBER_MEMORY,
                               oMEDICOAT_DATA_ARRAY => "DB16702_OPC_UA_MASTER_POWDER".UNIT_02.FEEDER_NOZZLE_LINE.NOZZLE_POWDER_FLOW);
   END_IF;
END_REGION
END_FUNCTION
